(* IEC 61131-3 sources: ironplc-benchmarks/compat_out (part 133) *)

(* revision History
hm	19. jan.2007	rev 1.1
	changed outputs to real to avoid overflow of integer
	added offset for better cascading of scale functions

hm	6. jan. 2008	rev 1.2
	improved performance

hm	26. oct. 2008	rev 1.3
	code optimization

hm	3. nov. 2008	rev 1.4
	used wrong factor in formula

*)
END_FUNCTION

(* @NESTEDCOMMENTS := 'Yes' *)
(* @PATH := '\/Engineering\/signal processing' *)
(* @OBJECTFLAGS := '0, 8' *)
(* @SYMFILEFLAGS := '2048' *)
FUNCTION SCALE_D : REAL
VAR_INPUT
	X : DWORD;
	I_LO : DWORD;
	I_HI : DWORD;
	O_LO : REAL;
	O_HI : REAL;
END_VAR

(*
version 1.2	11. jan. 2011
programmer 	hugo
tested by		oscat

Scale_D is used to translate and scale a DWORD input x to a real output.
the input is limited to I_LO <= X <= I_HI.

*)

(* @END_DECLARATION := '0' *)
IF I_HI = I_LO THEN
	SCALE_D := O_LO;
ELSE
	SCALE_D := (O_HI - O_LO) / DWORD_TO_REAL(I_HI - I_LO) * DWORD_TO_REAL(LIMIT(I_LO, X, I_HI) - I_LO) + O_LO;
END_IF;

(* revision history
hm	18. may. 2008	rev 1.0
	original version

hm	13. nov. 2008	rev 1.1
	corrected formula for negative gradient

hm	11. jan 2011	rev 1.2
	avoid division by 0
*)
END_FUNCTION

(* @NESTEDCOMMENTS := 'Yes' *)
(* @PATH := '\/Engineering\/signal processing' *)
(* @OBJECTFLAGS := '0, 8' *)
(* @SYMFILEFLAGS := '2048' *)
FUNCTION SCALE_R : REAL
VAR_INPUT
	X : REAL;
	I_LO : REAL;
	I_HI : REAL;
	O_LO : REAL;
	O_HI : REAL;
END_VAR

(*
version 1.2	11. jan. 2011
programmer 	hugo
tested by		oscat

Scale_R is used to translate and scale a REAL input x to a real output.
the input is limited to I_LO <= X <= I_HI.

*)

(* @END_DECLARATION := '0' *)
IF I_LO = I_HI THEN
	SCALE_R := O_LO;
ELSE
	SCALE_R := (O_HI - O_LO) / (I_HI - I_LO) * (LIMIT(I_LO, X, I_HI) - I_LO) + O_LO;
END_IF;

(* revision history
hm	18. may. 2008	rev 1.0
	original version

hm	13. nov. 2008	rev 1.1
	corrected formula for negative gradient

hm	11. jan 2011	rev 1.2
	avoid division by 0

*)
END_FUNCTION

(* @NESTEDCOMMENTS := 'Yes' *)
(* @PATH := '\/Engineering\/signal processing' *)
(* @OBJECTFLAGS := '0, 8' *)
(* @SYMFILEFLAGS := '2048' *)
FUNCTION SCALE_X2 : REAL
VAR_INPUT
	IN1: BOOL;
	IN2: BOOL;
	K : REAL;
	O : REAL;
END_VAR
VAR_INPUT (* CONSTANT *)
	IN1_MIN: REAL;
	IN1_MAX: REAL := 1000.0;
	IN2_MIN: REAL;
	IN2_MAX: REAL := 1000.0;
END_VAR

(*
version 1.1	26. oct. 2008
programmer 	hugo
tested by		tobias

	this functiob block can scale up to two inputs.
	the input can select between two values with true or false.
	the summed output is then scaled by an scale input K and a offset O can be added to the output.
	the min and max input configurations can be edited in the cfc editor by double clicking the symbol body.

*)

(* @END_DECLARATION := '0' *)
SCALE_X2 := (SEL(IN1, IN1_MIN, IN1_MAX)+ SEL(IN2, IN2_MIN, IN2_MAX)) * k + o;

(* revision history
hm	19. jan, 2007	rev 1.0
	original version

hm	26. oct. 2008	rev 1.1
	code optimized

*)
END_FUNCTION

(* @NESTEDCOMMENTS := 'Yes' *)
(* @PATH := '\/Engineering\/signal processing' *)
(* @OBJECTFLAGS := '0, 8' *)
(* @SYMFILEFLAGS := '2048' *)
FUNCTION SCALE_X4 : REAL
VAR_INPUT
	IN1: BOOL;
	IN2: BOOL;
	IN3: BOOL;
	IN4: BOOL;
	K : REAL;
	O : REAL;
END_VAR
VAR_INPUT (* CONSTANT *)
	IN1_MIN: REAL;
	IN1_MAX: REAL := 1000.0;
	IN2_MIN: REAL;
	IN2_MAX: REAL := 1000.0;
	IN3_MIN: REAL;
	IN3_MAX: REAL := 1000.0;
	IN4_MIN: REAL;
	IN4_MAX: REAL := 1000.0;
END_VAR

(*
version 1.1	26. oct. 2008
programmer 	hugo
tested by		tobias

	this function can scale up to 4 inputs.
	the input can select between two values with true or false.
	the summed output is then scaled by an scale input K and a offset O can be added to the output.
	the min and max input configurations can be edited in the cfc editor by double clicking the symbol body.

*)

(* @END_DECLARATION := '0' *)
SCALE_X4 := (SEL(IN1,IN1_MIN, IN1_MAX) + SEL(IN2, IN2_MIN, IN2_MAX)+SEL(IN3, IN3_MIN, IN3_MAX)+ SEL(IN4, IN4_MIN, IN4_MAX)) * k + o;

(* revision history
hm	19. jan. 2008	rev 1.0
	original version

hm	26. oct. 2008	rev 1.1
	optimized code
*)
END_FUNCTION

(* @NESTEDCOMMENTS := 'Yes' *)
(* @PATH := '\/Engineering\/signal processing' *)
(* @OBJECTFLAGS := '0, 8' *)
(* @SYMFILEFLAGS := '2048' *)
FUNCTION SCALE_X8 : REAL
VAR_INPUT
	in1: BOOL;
	in2: BOOL;
	in3: BOOL;
	in4: BOOL;
	in5: BOOL;
	in6: BOOL;
	in7: BOOL;
	in8: BOOL;
	K : REAL;
	O : REAL;
END_VAR
VAR_INPUT (* CONSTANT *)
	in1_min: REAL;
	in1_max: REAL := 1000.0;
	in2_min: REAL;
	in2_max: REAL := 1000.0;
	in3_min: REAL;
	in3_max: REAL := 1000.0;
	in4_min: REAL;
	in4_max: REAL := 1000.0;
	in5_min: REAL;
	in5_max: REAL := 1000.0;
	in6_min: REAL;
	in6_max: REAL := 1000.0;
	in7_min: REAL;
	in7_max: REAL := 1000.0;
	in8_min: REAL;
	in8_max: REAL := 1000.0;
END_VAR

(*
version 1.2	24. jan. 2009
programmer 	hugo
tested by	oscat

this function can scale up to 4 inputs.
the input can select between two values with true or false.
the summed output is then scaled by an scale input K and a offset O can be added to the output.
the min and max input configurations can be edited in the cfc editor by double clicking the symbol body.

*)

(* @END_DECLARATION := '0' *)
SCALE_X8 := (SEL(IN1,IN1_MIN, IN1_MAX)+ SEL(IN2,IN2_MIN, IN2_MAX)+SEL(IN3,IN3_MIN, IN3_MAX)+ SEL(IN4,IN4_MIN, IN4_MAX)
				+SEL(IN5,IN5_MIN, IN5_MAX)+ SEL(IN6,IN6_MIN, IN6_MAX)+SEL(IN7,IN7_MIN, IN7_MAX)+ SEL(IN8,IN8_MIN, IN8_MAX)) * k + o;

(* revision history
hm	19. jan. 2008	rev 1.0
	original version

hm	26. oct. 2008	rev 1.1
	optimized code

hm	24. jan. 2008	rev 1.2
	corrected error in formula
*)
END_FUNCTION

(* @NESTEDCOMMENTS := 'Yes' *)
(* @PATH := '\/Engineering\/signal processing' *)
(* @OBJECTFLAGS := '0, 8' *)
(* @SYMFILEFLAGS := '2048' *)
FUNCTION_BLOCK SEL2_OF_3
VAR_INPUT
	IN1 : REAL;
	IN2 : REAL;
	IN3 : REAL;
	D : REAL;
END_VAR
VAR_OUTPUT
	Y : REAL;
	W : INT;
	E : BOOL;
END_VAR
VAR
	D12: BOOL;
	D23: BOOL;
	D31: BOOL;
END_VAR

(*
	version 1.1	10. mar. 2009
	programmer 	oscat
	tested BY		oscat

SEL2_OF_3 checks if 3 input Signals are within a distance D from each other and calculates the average of the 3 inputs do not offset more than D from each other.
If 1 input is more than D greater or smaller than any other input it will be ignored and the average will be calcualted from the remaining 2 Inputs.
In the case the Output is only calculated from 2 Inputs a Warning Output W will display the Number of the discarded Input. if none of the 3 Inputs are within the allowed Delata D from each other,
an Error Output E is set True and the last valid Output will remain active until at least 2 Inputs are within a valid Range from each other.

*)

(* @END_DECLARATION := '0' *)
D12 := ABS(IN1-IN2) <= D;
D23 := ABS(IN2-IN3) <= D;
D31 := ABS(IN3-IN1) <= D;

IF (D12 AND D23) OR (D12 AND D31) OR (D23 AND D31) THEN
	(* all 3 inputs are valid *)
	Y := (IN1 + IN2 + IN3) * 0.333333333333;
	E := FALSE;
	W := 0;
ELSIF D12 THEN
	(* only inut 1 and 2 are valid *)
	Y := (In1 + IN2) * 0.5;
	E := FALSE;
	W := 3;
ELSIF D23 THEN
	(* only inut 2 and 3 are valid *)
	Y := (In2 + IN3) * 0.5;
	E := FALSE;
	W := 1;
ELSIF D31 THEN
	(* only inut 3 and 1 are valid *)
	Y := (In3 + IN1) * 0.5;
	E := FALSE;
	W := 2;
ELSE
	(* no calculation possible *)
	E := TRUE;
	W := 4;
END_IF;

(* revision history
hm	18. may 2008	rev 1.0
	original version

hm	10. mar. 2009	rev 1.1
	improved code
*)
END_FUNCTION_BLOCK

(* @NESTEDCOMMENTS := 'Yes' *)
(* @PATH := '\/Engineering\/signal processing' *)
(* @OBJECTFLAGS := '0, 8' *)
(* @SYMFILEFLAGS := '2048' *)
FUNCTION_BLOCK SEL2_OF_3B
VAR_INPUT
	IN1 : BOOL;
	IN2 : BOOL;
	IN3 : BOOL;
	TD : TIME;
END_VAR
VAR_OUTPUT
	Q : BOOL;
	W : BOOL;
END_VAR
VAR
	TDEL : TON;
END_VAR

(*
	version 1.0	19. may. 2008
	programmer 	oscat
	tested BY		oscat

SEL2_OF_3B is used to connect 3 binary sensors to one signal. the output Q reflects the state of at least two inputs.
if two or more of the 3 inputs ate TRUE then Q will be TRUE and if two or more of the three inputs are FALSE then Q will be false.
the main putrpose is the connection of 3 redundant binary sensors.
The output W will be active when one of the 3 inputs is of different state.
to avoid flickering while the sensors are switching the output W will become active after a programmed delay of TD.

*)

(* @END_DECLARATION := '0' *)
Q := (IN1 AND IN2) OR (IN1 AND IN3) OR (IN2 AND IN3);
TDEL(IN := (in1 XOR in2) OR (in1 XOR in3) OR (in2 XOR in3), PT := TD);
W := TDEL.Q;

(* revision history
hm		19. may 2008	rev 1.0
	original version

*)
END_FUNCTION_BLOCK

(* @NESTEDCOMMENTS := 'Yes' *)
(* @PATH := '\/Engineering\/signal processing' *)
(* @OBJECTFLAGS := '0, 8' *)
(* @SYMFILEFLAGS := '2048' *)
FUNCTION_BLOCK SH
VAR_INPUT
	in : REAL;
	CLK : BOOL;
END_VAR
VAR_OUTPUT
	out : REAL;
	trig : BOOL;
END_VAR
VAR
	edge : BOOL;
END_VAR

(*
version 1.1	16 jan 2007
programmer 	hugo
tested by		tobias

this sample and hold module samples an input at the rising edge of clk an stores it in out.
the out stays stable until the next rising clk edge appears.
a trigger output as active for one cycle when the output was updated.

*)
(* @END_DECLARATION := '0' *)
IF clk AND NOT edge THEN
	out := in;
	trig := TRUE;
ELSE;
	trig := FALSE;
END_IF;
edge := clk;

(* revision history

hm 16.1.2007	rev 1.1
	added trig output

*)
END_FUNCTION_BLOCK

(* @NESTEDCOMMENTS := 'Yes' *)
(* @PATH := '\/Engineering\/signal processing' *)
(* @OBJECTFLAGS := '0, 8' *)
(* @SYMFILEFLAGS := '2048' *)
FUNCTION_BLOCK SH_1
VAR_INPUT
	in : REAL;
	PT : TIME;
END_VAR
VAR_OUTPUT
	out : REAL;
	Trig : BOOL;
END_VAR
VAR
	last : TIME;
	tx: TIME;
END_VAR

(*
version 1.2	17 sep 2007
programmer 	hugo
tested by		tobias

this sample and hold module samples an input every PT seconds.
after a ample is taken the output Trig will be active for one cycle.

*)
(* @END_DECLARATION := '0' *)
(* read system time *)
tx := DWORD_TO_TIME(T_PLC_MS());

IF tx - last >= PT THEN
	last := tx;
	out := in;
	trig := TRUE;
ELSE
	trig := FALSE;
END_IF;

(* revision history

HM	6.1.2007	rev 1.1
	added trig output

HM	17.9.2007	rev 1.2
	replaced time() with T_PLC_MS() for compatibility reasons
*)

END_FUNCTION_BLOCK

(* @NESTEDCOMMENTS := 'Yes' *)
(* @PATH := '\/Engineering\/signal processing' *)
(* @OBJECTFLAGS := '0, 8' *)
(* @SYMFILEFLAGS := '2048' *)
FUNCTION_BLOCK SH_2
VAR_INPUT
	in : REAL;
	PT : TIME;
	N : INT := 16;
	disc : INT;
END_VAR
VAR_OUTPUT
	out : REAL;
	trig : BOOL;
	avg : REAL;
	high: REAL;
	low: REAL;
END_VAR
VAR
	M : INT;
	buf : ARRAY[0..15] OF REAL;
	buf2 : ARRAY[0..15] OF REAL;
	last : TIME;
	i : INT;
	start: INT;
	temp: REAL;
	stop: INT;
	tx: TIME;
	d2: INT;
END_VAR

(*
version 1.6	10. mar. 2009
programmer 	hugo
tested by		tobias

this sample and hold module samples an input every PT seconds.
this sample and hold also does avg and other calculations with the input data.
an average is calculated over N samples while for this calculation disc samples are discarded,
disc = 0 all samples are averaged,
if disc = 1 the lowest value is ignored,
if disc = 2 the lowest and highest values are ignored,
and so on.....

*)
(* @END_DECLARATION := '0' *)
(* read system time *)
tx := DWORD_TO_TIME(T_PLC_MS());
d2 := SHR(disc,1);

IF tx - last >= PT THEN
	last := tx;
	trig := TRUE;

	(* limit M to 0..16 *)
	M := LIMIT(1,N,16);

	(* edge detected lets take the sample *)
	FOR i := M - 1 TO 1 BY -1 DO buf2[i] := buf2[i-1]; END_FOR;
	buf2[0] := in;
	out := in;
	buf := buf2;

	(* sort the ARRAY lowest value AT 0 *)
	FOR start := 0 TO M - 2 DO
		FOR i := start+1 TO M - 1 DO
			IF buf[start] > buf[i] THEN
				temp := buf[start];
				buf[start] := buf[i];
				buf[i] := temp;
			END_IF;
		END_FOR;
	END_FOR;

	(* any calculation with the samples is here *)
	stop := M - 1 - d2;
	start := d2;
	IF NOT even(disc) THEN start := start + 1; END_IF;
	avg := 0;
	FOR i := start TO stop DO avg := avg + buf[i]; END_FOR;
	avg := avg / INT_TO_REAL(stop - start +1);
	low := buf[start];
	high := buf[stop];
ELSE
	Trig := FALSE;
END_IF;

(* revision history
hm 20. jan. 2007	rev 1.1
	added input N to specify the amout of samples for average and high low calculations
	added trig output

hm 10. sep. 2007 	rev 1.2
	an error would be generated if N was set to 0, now n is forced to1 if set to 0.
	index was out of array.

hm	17. sep. 2007	rev 1.3
	replaced time() with t_plc_ms() for compatibility reasons

hm	6. jan. 2008	rev 1.4
	improved performance

hm	14. jun. 2008	rev 1.5
	set default for input N = 16

hm	10. mar. 2009	rev 1.6
	added type conversion for compatibility reasons

*)
END_FUNCTION_BLOCK

(* @NESTEDCOMMENTS := 'Yes' *)
(* @PATH := '\/Engineering\/signal processing' *)
(* @OBJECTFLAGS := '0, 8' *)
(* @SYMFILEFLAGS := '2048' *)
FUNCTION_BLOCK SH_T
VAR_INPUT
	IN : REAL;
	E : BOOL;
END_VAR
VAR_OUTPUT
	OUT : REAL;
END_VAR

(*
version 1.1	18. oct. 2008
programmer 	hugo
tested by	oscat

this sample and hold module samples an input while en is high.
during the high time of en the output follows in.
the out stays stable until the en goes high again.
*)
(* @END_DECLARATION := '0' *)
IF E THEN out := in; END_IF;

(* revision history
hm	1. sep. 2006	rev 1.0
	original version

hm	18. oct. 2008	rev 1.1
	changed input en to e for compatibility reasons

*)
END_FUNCTION_BLOCK

(* @NESTEDCOMMENTS := 'Yes' *)
(* @PATH := '\/Engineering\/signal processing' *)
(* @OBJECTFLAGS := '0, 8' *)
(* @SYMFILEFLAGS := '2048' *)
FUNCTION STAIR : REAL
VAR_INPUT
	X : REAL;
	D : REAL;
END_VAR

(*
version 1.4	10. mar. 2009
programmer 	oscat
tested by		tobias

the function stair converts an anlog input signal to a staircase like output.
D is the step width for the output signal.
if D = 0 then the output follows the input without a chage.
*)
(* @END_DECLARATION := '0' *)
IF D > 0.0 THEN
	STAIR := DINT_TO_REAL(REAL_TO_DINT(X / D)) * D;
ELSE
	STAIR := X;
END_IF;

(* revision history
hm	28 jan 2007		rev 1.0
	original version

hm	27 dec 2007		rev 1.1
	changed code for better performance

hm	6. jan 2008		rev 1.2
	further performance improvement

hm	26. oct. 2008		rev 1.3
	optimized code

hm	10. mar. 2009	rev 1.4
	real constants updated to new systax using dot

*)
END_FUNCTION

(* @NESTEDCOMMENTS := 'Yes' *)
(* @PATH := '\/Engineering\/signal processing' *)
(* @OBJECTFLAGS := '0, 8' *)
(* @SYMFILEFLAGS := '2048' *)
FUNCTION_BLOCK STAIR2
VAR_INPUT
	X : REAL;
	D : REAL;
END_VAR
VAR_OUTPUT
	Y: REAL;
END_VAR

(*
version 1.4	10. mar. 2009
programmer 	hugo
tested by		oscat

the function stair2 converts an anlog input signal to a staircase like output.
D is the step width for the output signal. the output will use D as a hysteresis for a stairchange.
if D = 0 then the output follows the input without a chage.
*)
(* @END_DECLARATION := '0' *)
IF D > 0.0 THEN
	IF X >= Y + D OR X <= Y - D THEN Y := FLOOR(X/D) * D; END_IF;
ELSE
	Y := X;
END_IF;

(* revision history
hm	28 jan 2007		rev 1.0
	original version

hm	27. dec 2007	rev 1.1
	changed code for better performance

hm	30. jun. 2008	rev 1.2
	added type conversions to avoid warnings under codesys 3.0

ks	26. oct. 2008	rev 1.3
	improved code

hm	10. mar. 2009	rev 1.4
	real constants updated to new systax using dot

*)
END_FUNCTION_BLOCK

(* @NESTEDCOMMENTS := 'Yes' *)
(* @PATH := '\/Engineering\/signal processing' *)
(* @OBJECTFLAGS := '0, 8' *)
(* @SYMFILEFLAGS := '2048' *)
FUNCTION_BLOCK TREND
VAR_INPUT
	X : REAL;
END_VAR
VAR_OUTPUT
	Q : BOOL;
	TU : BOOL;
	TD : BOOL;
	D : REAL;
END_VAR
VAR
	last_X: REAL;
END_VAR

(*
version 1.0	21. aug. 2009
programmer 	hugo
tested by		oscat

trend analyses the trend of a input signal.
The Output Q is True if the input X is >= last_X and is false if the input X is <= last_X
in addition to the trend the output TU will be high for one cycle to signal a rising of the input value X
and  TD will signal a decreasing value on the input X.
in case of a change the output D will show the delta of the input to the last input value.

*)
(* @END_DECLARATION := '0' *)
TU := X > last_X;
TD := X < last_X;
Q := TU OR TD;
D := X - LAST_X;

last_X := X;

(* revision history
hm	21. aug. 2009	rev 1.0
	original version

*)

END_FUNCTION_BLOCK

(* @NESTEDCOMMENTS := 'Yes' *)
(* @PATH := '\/Engineering\/signal processing' *)
(* @OBJECTFLAGS := '0, 8' *)
(* @SYMFILEFLAGS := '2048' *)
FUNCTION_BLOCK TREND_DW
VAR_INPUT
	X : DWORD;
END_VAR
VAR_OUTPUT
	Q : BOOL;
	TU : BOOL;
	TD : BOOL;
	D : DWORD;
END_VAR
VAR
	last_X: DWORD;
END_VAR

(*
version 1.2	14. mar. 2009
programmer 	hugo
tested by		oscat

trend_DW analyses the trend of a input signal.
The Output Q is True if the input X is >= last_X and is false if the input X is <= last_X
in addition to the trend the output TU will be high for one cycle to signal a rising of the input value X
and  TD will signal a decreasing value on the input X.
in case of a change the output D will show the delta of the input to the last input value.

*)
(* @END_DECLARATION := '0' *)
IF X > last_X THEN
	TU := TRUE;
	TD := FALSE;
	D := X - last_X;
	Q := TRUE;
ELSIF X < last_X THEN
	TD := TRUE;
	TU := FALSE;
	D := last_X - X;
	Q := FALSE;
ELSE
	TU := FALSE;
	TD := FALSE;
	D := 0;
END_IF;
last_X := X;

(* revision history
hm	21. nov. 2008	rev 1.0
	original version

hm	20. feb. 2009	rev 1.1
	added outputs TU, TD and D

hm	14. mar. 2009	rev 1.2
	removed double assignments

*)

END_FUNCTION_BLOCK

(* @NESTEDCOMMENTS := 'Yes' *)
(* @PATH := '\/Engineering\/signal processing' *)
(* @OBJECTFLAGS := '0, 8' *)
(* @SYMFILEFLAGS := '2048' *)
FUNCTION WORD_TO_RANGE : REAL
VAR_INPUT
	X : WORD;
	low : REAL;
	high : REAL;
END_VAR

(*
version 1.1	10. mar. 2009
programmer 	hugo
tested by		tobias

Word_to_Range converts a Byte into a real between low and high.

*)
(* @END_DECLARATION := '0' *)
WORD_TO_RANGE := (high - low) * WORD_TO_REAL(X) * 0.00001525902189669640 + low;

(* revision history
hm	9. jan 2008	rev 1.0
	original version

hm	10. mar. 2009	rev 1.1
	improved code
*)

END_FUNCTION

(* @NESTEDCOMMENTS := 'Yes' *)
(* @PATH := '\/List Processing' *)
(* @OBJECTFLAGS := '0, 8' *)
(* @SYMFILEFLAGS := '2048' *)
FUNCTION LIST_ADD : BOOL
VAR_INPUT
	SEP : BYTE;
	INS : STRING[LIST_LENGTH];
END_VAR
VAR_IN_OUT
	LIST : STRING[LIST_LENGTH];
END_VAR
VAR
	sx : STRING[1];
END_VAR

(*
version 2.0		21. mar. 2011
programmer 	hugo
tested by		kurt

LIST_ADD h�ngt ein weiteres element ans ende einer liste.
die liste liegt als string von elementen vor die mit den zeichen SEP am anfang makiert sind.

*)
(* @END_DECLARATION := '0' *)
sx := CHR_TO_STRING(SEP);			(* convert separation character to string *)
INS := CONCAT(sx, INS);					(* start element with separation character *)

IF LEN(LIST) + LEN(INS) > LIST_LENGTH THEN
	LIST_ADD := FALSE;					(* return false if element does not fit *)
ELSE
	LIST := CONCAT(LIST, INS);
	LIST_ADD := TRUE;
END_IF;

(* revision histroy

hm	21. mar. 2011	rev 2.0
	original release
*)

END_FUNCTION

(* @NESTEDCOMMENTS := 'Yes' *)
(* @PATH := '\/List Processing' *)
(* @OBJECTFLAGS := '0, 8' *)
(* @SYMFILEFLAGS := '2048' *)
FUNCTION LIST_CLEAN : BOOL
VAR_INPUT
	SEP : BYTE;
END_VAR
VAR_IN_OUT
	LIST : STRING[LIST_LENGTH];
END_VAR
VAR
	pt : REF_TO ARRAY[1..LIST_LENGTH] OF BYTE;
	read : INT := 1;
	write : INT := 1;
	last: BYTE;
	c: BYTE;
END_VAR

(*
version 2.0	21. mar. 2011
programmer 	hugo
tested by		oscat

LIST_CLEAN bereinigt eine liste von leeren Elementen.
die liste liegt als string von elementen vor die mit den zeichen SEP am anfang markiert sind.

*)
(* @END_DECLARATION := '0' *)
pt := REF(LIST);

FOR read := 1 TO LIST_LENGTH DO
	c := pt^[read];								(* read character from list *)
	IF c = 0 THEN EXIT;						(* exit the loop if character definbes end of string *)
	ELSIF c <> SEP OR sep <> last THEN	(* copy element from read to write position unless a double sep character is present *)
		pt^[write] := c;
		write := write + 1;
	END_IF;
	last := c;									(* remember last character *)
END_FOR;

IF last = SEP THEN write := write - 1; END_IF;		(* if last character is sep then delete empty element at end *)
IF write <= STRING_LENGTH THEN pt^[write] := 0;	 END_IF;		(* terminate string with 0 *)

LIST_CLEAN := TRUE;						(* retrun TRUE *)

(* revision histroy
hm	28. jun. 2008	rev 1.0
	original release

hm	19. jan. 2011	rev 1.1
	changed STRING[255] to STRING[LIST_LENGTH]

hm	21. mar. 2011	rev 2.0
	all elements start with SEP

*)

END_FUNCTION

(* @NESTEDCOMMENTS := 'Yes' *)
(* @PATH := '\/List Processing' *)
(* @OBJECTFLAGS := '0, 8' *)
(* @SYMFILEFLAGS := '2048' *)
FUNCTION LIST_GET : STRING[LIST_LENGTH]
VAR_INPUT
	SEP : BYTE;
	POS : INT;
END_VAR
VAR_IN_OUT
	LIST : STRING[LIST_LENGTH];
END_VAR
VAR
	i : INT := 1;
	o : INT := 1;
	pt : REF_TO ARRAY[1..LIST_LENGTH] OF BYTE;
	po : REF_TO ARRAY[1..LIST_LENGTH] OF BYTE;
	cnt: INT := 0;
	c: BYTE;
END_VAR

(*
version 2.0	21. mar. 2011
programmer 	hugo
tested by		oscat

LIST_GET liefert das element an der stelle pos einer liste.
die liste liegt als string von elementen vor die mit den zeichen SEP am anfang makiert sind.

*)
(* @END_DECLARATION := '0' *)
pt := REF(LIST);							(* load pointers *)
po := REF(LIST_GET);

REPEAT
	c := pt^[i];
	IF cnt = pos THEN						(* copy element to output string *)
		IF c = SEP  THEN EXIT; END_IF;		(* next element stop copy and finish *)
		po^[o] := c;
		o := o + 1;
	ELSIF c = SEP THEN
		cnt := cnt + 1;
	END_IF;
	i := i + 1;
UNTIL
	(i = LIST_LENGTH) OR (c = 0)
END_REPEAT;
po^[o] := 0;						(* close the output string *)

(* revision histroy
hm	20. jun. 2008	rev 1.0
	original release

hm	19. jan. 2011	rev 1.1
	changed STRING[255] to strring(LIST_LENGTH)

hm	21. mar. 2011	rev 2.0
	all list elements start with SEP
*)

END_FUNCTION

(* @NESTEDCOMMENTS := 'Yes' *)
(* @PATH := '\/List Processing' *)
(* @OBJECTFLAGS := '0, 8' *)
(* @SYMFILEFLAGS := '2048' *)
FUNCTION LIST_INSERT : BOOL
VAR_INPUT
	SEP : BYTE;
	POS : INT;
	INS : STRING[LIST_LENGTH];
END_VAR
VAR_IN_OUT
	LIST : STRING[LIST_LENGTH];
END_VAR
VAR
	pt : REF_TO ARRAY[1..LIST_LENGTH] OF BYTE;
	read : INT := 1;
	cnt : INT := 1;
	sx : STRING[1];
END_VAR

(*
version 2.0	21. mar. 2011
programmer 	hugo
tested by		oscat

LIST_INSERT setzt ein element an der stelle pos in eine liste ein.
die liste liegt als string von elementen vor die mit den zeichen SEP am anfang markiert sind.

*)
(* @END_DECLARATION := '0' *)
(* load pointers *)
pt := REF(LIST);

IF LEN(ins) + 1 + LEN(LIST) > LIST_LENGTH THEN
	LIST_INSERT := FALSE;
ELSE
	LIST_INSERT := TRUE;
	(* search for position *)
	WHILE read < LIST_LENGTH DO
		IF cnt >= POS THEN
			sx := CHR_TO_STRING(SEP);
			INS := CONCAT(sx, INS);
			LIST := INSERT(LIST, INS, read - 1);
			LIST_INSERT := TRUE;
			RETURN;
		END_IF;
		IF pt^[read]  = 0 THEN				(* list is too short add empty element *)
			pt^[read] := SEP;
			pt^[read + 1] := 0;
		END_IF;
		read := read + 1;
		IF pt^[read] = SEP OR pt^[read] = 0 THEN cnt := cnt + 1; END_IF;
	END_WHILE;
END_IF;

(* revision histroy
hm	28. jun. 2008	rev 1.0
	original release

hm	17. dec. 2008	rev 1.1
	changes name of function chr to chr_to_string

hm	19. jan. 2011	rev 1.2
	changed STRING[255] to STRING[LIST_LENGTH]

hm	21. mar. 2011	rev 2.0
	all list elements start with SEP

*)

END_FUNCTION

(* @NESTEDCOMMENTS := 'Yes' *)
(* @PATH := '\/List Processing' *)
(* @OBJECTFLAGS := '0, 8' *)
(* @SYMFILEFLAGS := '2048' *)
FUNCTION LIST_LEN : INT
VAR_INPUT
	SEP : BYTE;
END_VAR
VAR_IN_OUT
	LIST : STRING[LIST_LENGTH];
END_VAR
VAR
	pt : REF_TO ARRAY[1..LIST_LENGTH] OF BYTE;
	pos: INT := 1;
	c: BYTE;
END_VAR

(*
version 2.0	21. mar. 2011
programmer 	hugo
tested by		oscat

LIST_LEN liefert die anzahl der elemente einer liste.
die liste liegt als string von elementen vor die mit den zeichen SEP am anfang markiert sind.

*)
(* @END_DECLARATION := '0' *)
pt := REF(LIST);
LIST_LEN := 0;
REPEAT
	c := pt^[pos];
	IF c = SEP THEN LIST_LEN := LIST_LEN + 1; END_IF;
	pos := pos + 1;
UNTIL
	c = 0 OR pos > LIST_LENGTH
END_REPEAT;

(* revision histroy
hm	25. jun. 2008	rev 1.0
	original release

hm	16. oct. 2008	rev 1.1
	fixed a problem where list_len would only work up to LIST_LENGTH

hm	19. jan. 2001	rev 1.2
	changed STRING[255] to STRING[LIST_LENGTH]

hm	21. mar. 2011	rev 2.0
	all list elements start with SEP

*)

END_FUNCTION

(* @NESTEDCOMMENTS := 'Yes' *)
(* @PATH := '\/List Processing' *)
(* @OBJECTFLAGS := '0, 8' *)
(* @SYMFILEFLAGS := '2048' *)
FUNCTION_BLOCK LIST_NEXT
VAR_INPUT
	SEP : BYTE;
	RST : BOOL;
END_VAR
VAR_IN_OUT
	LIST : STRING[LIST_LENGTH];
END_VAR
VAR_OUTPUT
	LEL : STRING[LIST_LENGTH];
	NUL : BOOL;
END_VAR
VAR
	pos : INT := 1;
	pt : REF_TO ARRAY[1..LIST_LENGTH] OF BYTE;
	po : REF_TO ARRAY[1..LIST_LENGTH] OF BYTE;
	c: BYTE;
	write: INT;
END_VAR

(*
version 2.0	21. mar. 2011
programmer 	hugo
tested by		oscat

LIST_NEXT retrieves the next element of a list, starting from element 1 after reset or first init.
when the end of the lisat is reached a '' empty string is returned and NUL is set to true.
die liste liegt als string von elementen vor die mit den zeichen SEP am anfang markiert sind.

*)
(* @END_DECLARATION := '0' *)
pt := REF(LIST);
po := REF(LEL);

IF rst THEN
	pos := 1;
END_IF;

IF pt^[pos] = 0 OR pos = LIST_LENGTH THEN
	LEL := '';
	NUL := TRUE;
ELSE
	NUL := FALSE;
	write := 1;
	FOR pos := pos + 1 TO LIST_LENGTH DO
		c := pt^[pos];
		IF c = 0 OR c = SEP THEN
			po^[write] := 0;
			RETURN;
		ELSE
			po^[write] := pt^[pos];
			write := write + 1;
		END_IF;
	END_FOR;
END_IF;

(* revision histroy
hm	25. jun. 2008	rev 1.0
	original release

hm	19. jan. 2011	rev 1.1
	changed STRING[255] to STRING[LIST_LENGTH]

hm	21. mar. 2011	rev 2.0
	all elements start with SEP

*)

END_FUNCTION_BLOCK

(* @NESTEDCOMMENTS := 'Yes' *)
(* @PATH := '\/List Processing' *)
(* @OBJECTFLAGS := '0, 8' *)
(* @SYMFILEFLAGS := '2048' *)
FUNCTION LIST_RETRIEVE : STRING[LIST_LENGTH]
VAR_INPUT
	SEP : BYTE;
	POS : INT;
END_VAR
VAR_IN_OUT
	LIST : STRING[LIST_LENGTH];
END_VAR
VAR
	i :	INT;
	o : INT := 1;
	w : INT := 1;
	pt : REF_TO ARRAY[1..LIST_LENGTH] OF BYTE;
	po : REF_TO ARRAY[1..LIST_LENGTH] OF BYTE;
	cnt: INT := 0;
	c: BYTE;
END_VAR

(*
version 2.0		21. mar. 2011
programmer 	hugo
tested by		oscat

LIST_RETRIEVE liefert das element an der stelle pos einer liste und l�scht das element aus der liste.
die liste liegt als string von elementen vor die mit den zeichen SEP separiert sind.

*)
(* @END_DECLARATION := '0' *)
(* load pointers *)
pt := REF(LIST);
po := REF(LIST_RETRIEVE);

IF pos > 0 THEN
	FOR i := 1 TO LIST_LENGTH DO
		c := pt^[i];
		IF c = 0 THEN
			po^[o] := 0;
			IF cnt < pos THEN pt^[w + 1] := 0; ELSE pt^[w] := 0; END_IF;
			RETURN;
		ELSIF cnt = pos AND c <> SEP THEN				(* we have found the element *)
			po^[o] := pt^[i];
			o := o + 1;
		ELSIF cnt >= pos THEN
			pt^[w] := c;
			w := w + 1;
		ELSE
			w := i;
		END_IF;
		IF c = sep THEN cnt := cnt + 1; END_IF;
	END_FOR;
ELSE
	LIST_RETRIEVE := '';
END_IF;

(* revision histroy
hm	28. jun. 2008	rev 1.0
	original release

hm	19. jan. 2011	rev 1.1
	changed STRING[255] to STRING[LIST_LENGTH]

hm	21. mar. 2011	rev 2.0
	all elements start with SEP
*)

END_FUNCTION

(* @NESTEDCOMMENTS := 'Yes' *)
(* @PATH := '\/List Processing' *)
(* @OBJECTFLAGS := '0, 8' *)
(* @SYMFILEFLAGS := '2048' *)
FUNCTION LIST_RETRIEVE_LAST : STRING[LIST_LENGTH]
VAR_INPUT
	SEP : BYTE;
END_VAR
VAR_IN_OUT
	LIST : STRING[LIST_LENGTH];
END_VAR
VAR
	i :	INT;
	last : INT := 1;
	pt : REF_TO ARRAY[1..LIST_LENGTH] OF BYTE;
	c: BYTE;
END_VAR

(*
version 2.0		21. mar. 2011
programmer 	hugo
tested by		oscat

LIST_RETRIEVE_LAST liefert das letzte element einer liste und l�scht das element aus der liste.
die liste liegt als string von elementen vor die mit den zeichen SEP beginnen.

*)
(* @END_DECLARATION := '0' *)
(* load pointers *)
pt := REF(LIST);

(* search position of last element *)
FOR i := 1 TO LIST_LENGTH DO
	c := pt^[i];
	IF c = 0 THEN
		EXIT;
	ELSIF C = SEP THEN
		last := i;
	END_IF;
END_FOR;
(* return last element of list *)
/* LIST_RETRIEVE_LAST := MID(LIST, LIST_LENGTH, last + 1); */
(* terminate list at i *)
pt^[last] := 0;

(* revision histroy
hm	21. mar. 2011	rev 2.0
	new module
*)
END_FUNCTION

(* @NESTEDCOMMENTS := 'Yes' *)
(* @PATH := '\/Logic\/FF edge triggered' *)
(* @OBJECTFLAGS := '0, 8' *)
(* @SYMFILEFLAGS := '2048' *)
FUNCTION_BLOCK COUNT_BR
VAR_INPUT
	SET0 : BOOL;
	IN : BYTE;
	UP : BOOL;
	DN : BOOL;
	STEP : BYTE := 1;
	MX : BYTE := 255;
	RST : BOOL;
END_VAR
VAR_OUTPUT
	CNT : BYTE;
END_VAR
VAR
	last_up: BOOL;
	last_dn: BOOL;
END_VAR

(*
	version 1.0	16 jan 2008
	programmer 	hugo
	tested BY	tobias

Count_BR is a byte counter with independen up and dn inputs. the counter counts from 0 to mx and continues at 0 after is has reached mx
a step input sets the counters stepping width.

*)
(* @END_DECLARATION := '0' *)
IF rst THEN
	cnt := 0;
ELSIF set0 THEN
	cnt := LIMIT(0,in,mx);
ELSIF up AND NOT last_up THEN
	cnt := INT_TO_BYTE(INC(cnt,step,mx));
ELSIF dn AND NOT last_dn THEN
	cnt := INT_TO_BYTE(inc(cnt,-step,mx));
END_IF;
last_up := up;
last_dn := dn;

(* revision history
hm	16. jan 2008	rev 1.0
	original version

*)
END_FUNCTION_BLOCK

(* @NESTEDCOMMENTS := 'Yes' *)
(* @PATH := '\/Logic\/FF edge triggered' *)
(* @OBJECTFLAGS := '0, 8' *)
(* @SYMFILEFLAGS := '2048' *)
FUNCTION_BLOCK COUNT_DR
VAR_INPUT
	SET0 : BOOL;
	IN : DWORD;
	UP : BOOL;
	DN : BOOL;
	STEP : DWORD := 1;
	MX : DWORD := 16#FFFFFFFF;
	RST : BOOL;
END_VAR
VAR_OUTPUT
	CNT : DWORD;
END_VAR
VAR
	last_up: BOOL;
	last_dn: BOOL;
END_VAR

(*
	version 1.1	20. jan. 2011
	programmer 	hugo
	tested BY		tobias

Count_DR is a DWORD counter with independen up and dn inputs. the counter counts from 0 to mx and continues at 0 after is has reached mx
a step input sets the counters stepping width.

*)
(* @END_DECLARATION := '0' *)
IF rst THEN
	cnt := 0;
ELSIF set0 THEN
	cnt := LIMIT(0,in,mx);
ELSIF up AND NOT last_up THEN
	IF STEP > MX - CNT THEN
		CNT := CNT - MX + STEP - 1;
	ELSE
		CNT := CNT + STEP;
	END_IF;
ELSIF dn AND NOT last_dn THEN
	IF STEP > CNT THEN
		CNT := CNT - STEP + MX + 1;
	ELSE
		CNT := CNT - STEP;
	END_IF;
END_IF;
last_up := up;
last_dn := dn;

(* revision history
hm	12. jun 2008	rev 1.0
	original version

hm	20. jan. 2011	rev 1.1
	corrected init value of MX to 16#FFFFFFFF

*)
END_FUNCTION_BLOCK

(* @NESTEDCOMMENTS := 'Yes' *)
(* @PATH := '\/Logic\/FF edge triggered' *)
(* @OBJECTFLAGS := '0, 8' *)
(* @SYMFILEFLAGS := '2048' *)
FUNCTION_BLOCK FF_D2E
VAR_INPUT
	D0 : BOOL;
	D1 : BOOL;
	CLK : BOOL;
	RST : BOOL;
END_VAR
VAR_OUTPUT
	Q0 : BOOL;
	Q1 : BOOL;
END_VAR
VAR
	edge : BOOL;
END_VAR

(*
version 1.3	14. mar. 2009
programmer 	hugo
tested by		oscat

dual D-type flip flop with reset and rising clock trigger

*)

(* @END_DECLARATION := '0' *)
IF rst THEN
	Q0 := FALSE;
	Q1 := FALSE;
ELSIF clk AND NOT edge THEN
	Q0 := D0;
	Q1 := D1;
END_IF;
edge := CLK;

(* revision history
hm	25. dec 2007	rev 1.0
	original version

hm	27. dec 2007	rev 1.1
	changed code for better performance

hm	30. oct. 200	rev 1.2
	deleted unnecessary init with 0

hm	14. mar. 2009	rev 1.3
	removed double assignments

*)

END_FUNCTION_BLOCK

(* @NESTEDCOMMENTS := 'Yes' *)
(* @PATH := '\/Logic\/FF edge triggered' *)
(* @OBJECTFLAGS := '0, 8' *)
(* @SYMFILEFLAGS := '2048' *)
FUNCTION_BLOCK FF_D4E
VAR_INPUT
	D0 : BOOL;
	D1 : BOOL;
	D2 : BOOL;
	D3 : BOOL;
	CLK : BOOL;
	RST : BOOL;
END_VAR
VAR_OUTPUT
	Q0 : BOOL;
	Q1 : BOOL;
	Q2 : BOOL;
	Q3 : BOOL;
END_VAR
VAR
	edge : BOOL;
END_VAR

(*
version 1.3	14. mar. 2009
programmer 	hugo
tested by		oscat

quad D-type flip flop with reset and rising clock trigger

*)

(* @END_DECLARATION := '0' *)
IF rst THEN
	Q0 := FALSE;
	Q1 := FALSE;
	Q2 := FALSE;
	Q3 := FALSE;
ELSIF clk AND NOT edge THEN
	Q0 := D0;
	Q1 := D1;
	Q2 := D2;
	Q3 := D3;
END_IF;
edge := CLK;

(* revision history
hm	4. aug 2006	rev 1.0
	original version

hm	27. dec 2007	rev 1.1
	changed code for better performance

hm	30. oct. 200	rev 1.2
	deleted unnecessary init with 0

hm	14. mar. 2009	rev 1.3
	removed double assignments

*)

END_FUNCTION_BLOCK

(* @NESTEDCOMMENTS := 'Yes' *)
(* @PATH := '\/Logic\/FF edge triggered' *)
(* @OBJECTFLAGS := '0, 8' *)
(* @SYMFILEFLAGS := '2048' *)
FUNCTION_BLOCK FF_DRE
VAR_INPUT
	SET0 : BOOL;
	D : BOOL;
	CLK : BOOL;
	RST : BOOL;
END_VAR
VAR_OUTPUT
	Q : BOOL;
END_VAR
VAR
	edge : BOOL;
END_VAR

(*
version 1.2	30. oct. 2008
programmer 	hugo
tested by	oscat

D-type flip flop with set, reset and rising clock trigger

*)

(* @END_DECLARATION := '0' *)
IF rst OR set0 THEN
	Q := NOT rst;
ELSIF clk AND NOT edge THEN
	Q := D;
END_IF;
edge := CLK;

(* revision history
hm	4. aug 2006		rev 1.0
	original version

hm	27. dec 2007	rev 1.1
	changed code for better performance

hm	30. oct. 2008	rev 1.2
	optimized performance
*)
END_FUNCTION_BLOCK

(* @NESTEDCOMMENTS := 'Yes' *)
(* @PATH := '\/Logic\/FF edge triggered' *)
(* @OBJECTFLAGS := '0, 8' *)
(* @SYMFILEFLAGS := '2048' *)
FUNCTION_BLOCK FF_JKE
VAR_INPUT
	SET0 : BOOL;
	J : BOOL;
	CLK : BOOL;
	K : BOOL;
	RST : BOOL;
END_VAR
VAR_OUTPUT
	Q : BOOL;
END_VAR
VAR
	edge : BOOL;
END_VAR

(*
version 1.2	30. oct. 2008
programmer 	hugo
tested by	oscat

JK-type flip flop with set, reset and rising clock trigger
set and reset are asynchron while the FF is rising edge triggered
J=0 and K=0 and CLK >>> no action
J=1 and K=0 and CLK >>> output = 1
J=0 and K=1 and CLK >>> output = 0
J=1 and K=1 and CLK >>> toggle output

*)

(* @END_DECLARATION := '0' *)
IF rst OR set0 THEN
	Q := NOT rst;
ELSIF clk AND NOT edge THEN
	IF J XOR K THEN Q := J;
	ELSE Q := K XOR Q;
	END_IF;
END_IF;
edge := CLK;

(* revision history
hm	4. aug 2006		rev 1.0
	original version

hm	27. dec 2007	rev 1.1
	changed code for better performance

hm	30. oct. 2008	rev 1.2
	optimized performance
*)
END_FUNCTION_BLOCK

(* @NESTEDCOMMENTS := 'Yes' *)
(* @PATH := '\/Logic\/FF edge triggered' *)
(* @OBJECTFLAGS := '0, 8' *)
(* @SYMFILEFLAGS := '2048' *)
FUNCTION_BLOCK FF_RSE
VAR_INPUT
	CS : BOOL;
	CR : BOOL;
	RST : BOOL;
END_VAR
VAR_OUTPUT
	Q : BOOL;
END_VAR
VAR
	es, er : BOOL;
END_VAR

(*
version 1.0	16. jul. 2008
programmer 	hugo
tested by	oscat

this is a rising edge triggered rs flip flop
a rising edge on CS sets Q = TRUE and a rising edge on CR sets Q = FALSE.
CR has priority over CS.

*)

(* @END_DECLARATION := '0' *)
IF rst THEN
	(* asynchronous reset *)
	Q := FALSE;
ELSIF CR AND NOT er THEN
	(* rising edge on CR *)
	Q := FALSE;
ELSIF CS AND NOT es THEN
	(* rising edge on CS *)
	Q := TRUE;
END_IF;

es := CS;
er := CR;

(* revision history

hm	16. jul. 2008	rev 1.0
	original version

*)

END_FUNCTION_BLOCK

(* @NESTEDCOMMENTS := 'Yes' *)
(* @PATH := '\/Logic\/FF edge triggered' *)
(* @OBJECTFLAGS := '0, 8' *)
(* @SYMFILEFLAGS := '2048' *)
FUNCTION_BLOCK SELECT_8
VAR_INPUT
	E : BOOL;
	SET0 : BOOL;
	IN : BYTE;
	UP : BOOL;
	DN : BOOL;
	RST : BOOL;
END_VAR
VAR_OUTPUT
	Q0, Q1, Q2, Q3, Q4, Q5, Q6, Q7 : BOOL;
	STATE : INT;
END_VAR
VAR
	last_up: BOOL;
	last_dn : BOOL;
END_VAR

(*
	version 1.1	27. feb. 2009
	programmer 	hugo
	tested BY		oscat

select_8 selects one of 8 outputs at any time. the outputscan be selected by up or down keys and an independent anable switches all outouts off if set false

*)
(* @END_DECLARATION := '0' *)
IF rst THEN
	state := 0;
ELSIF set0 THEN
	state := IN;
ELSIF up AND NOT last_up THEN
	state := inc(state,1,7);
ELSIF dn AND NOT last_dn THEN
	state := inc(state,-1,7);
END_IF;
last_UP := UP;
last_DN := DN;

Q0 := FALSE;
Q1 := FALSE;
Q2 := FALSE;
Q3 := FALSE;
Q4 := FALSE;
Q5 := FALSE;
Q6 := FALSE;
Q7 := FALSE;

IF E THEN
	CASE state OF
		0: Q0 := TRUE;
		1: Q1 := TRUE;
		2: Q2 := TRUE;
		3: Q3 := TRUE;
		4: Q4 := TRUE;
		5: Q5 := TRUE;
		6: Q6 := TRUE;
		7: Q7 := TRUE;
	END_CASE;
END_IF;

(* revision history
hm	16. jan 2008	rev 1.0
	original version

hm	27. feb. 2009	rev 1.1
	renamed input en to e
*)
END_FUNCTION_BLOCK

(* @NESTEDCOMMENTS := 'Yes' *)
(* @PATH := '\/Logic\/FF edge triggered' *)
(* @OBJECTFLAGS := '0, 8' *)
(* @SYMFILEFLAGS := '2048' *)
FUNCTION_BLOCK SHR_4E
VAR_INPUT
	SET0 : BOOL;
	D0: BOOL;
	CLK: BOOL;
	RST: BOOL;
END_VAR
VAR_OUTPUT
	Q0: BOOL;
	Q1: BOOL;
	Q2: BOOL;
	Q3: BOOL;
END_VAR
VAR
	trig : R_TRIG;
END_VAR

(*
version 1.1	25. oct. 2008
programmer 	hugo
tested by		tobias

4 bit shift register with reset

*)
(* @END_DECLARATION := '0' *)
(* trig.Q signals a rising edge on clk *)
trig(clk := clk);

IF set0 OR rst THEN
	Q0 := NOT rst;
	Q1 := Q0;
	Q2 := Q0;
	Q3 := Q0;
ELSIF trig.Q THEN
	Q3 := Q2;
	Q2 := Q1;
	Q1 := Q0;
	Q0 := D0;
END_IF;

(* revision history
hm	4. aug. 2006	rev 1.0
	original version

hm	25. oct. 2008	rev 1.1
	optimized code

*)
END_FUNCTION_BLOCK

(* @NESTEDCOMMENTS := 'Yes' *)
(* @PATH := '\/Logic\/FF edge triggered' *)
(* @OBJECTFLAGS := '0, 8' *)
(* @SYMFILEFLAGS := '2048' *)
FUNCTION_BLOCK SHR_4UDE
VAR_INPUT
	SET0 : BOOL;
	D0: BOOL;
	D3: BOOL;
	CLK: BOOL;
	DN : BOOL;
	RST: BOOL;

END_VAR
VAR_OUTPUT
	Q0: BOOL;
	Q1: BOOL;
	Q2: BOOL;
	Q3: BOOL;
END_VAR
VAR
	trig : R_TRIG;
END_VAR

(*
version 1.2	14. mar. 2009
programmer 	hugo
tested by		tobias

4 bit shift register with reset up / down direction input

*)
(* @END_DECLARATION := '0' *)
(* trig.Q signals a rising edge on clk *)
trig(clk := clk);

IF set0 OR rst THEN
	Q0 := NOT RST;
	Q1 := Q0;
	Q2 := Q0;
	Q3 := Q0;
ELSIF trig.Q THEN
	IF dn THEN
		Q0 := Q1;
		Q1 := Q2;
		Q2 := Q3;
		Q3 := D3;
	ELSE
		Q3 := Q2;
		Q2 := Q1;
		Q1 := Q0;
		Q0 := D0;
	END_IF;
END_IF;

(* revision history
hm	4. aug. 2006	rev 1.0
	original version

hm	25. oct. 2008	rev 1.1
	optimized code

hm	14. mar. 2009	rev 1.2
	removed double assignments

*)
END_FUNCTION_BLOCK

(* @NESTEDCOMMENTS := 'Yes' *)
(* @PATH := '\/Logic\/FF edge triggered' *)
(* @OBJECTFLAGS := '0, 8' *)
(* @SYMFILEFLAGS := '2048' *)
FUNCTION_BLOCK SHR_8PLE
VAR_INPUT
	Din : BOOL;
	Dload : BYTE;
	CLK: BOOL;
	UP: BOOL :=1;
	load : BOOL;
	RST: BOOL;
END_VAR
VAR_OUTPUT
	DOut: BOOL;
END_VAR
VAR
	edge : BOOL :=1;
	register : BYTE;
END_VAR

(*
version 1.0	4 aug 2006
programmer 	hugo
tested by	oscat

8 bit shift register with reset and parallel load
the register can shift up or down
it also has a serial input.
the Din input is on Bit0 for up shift and on bit 7 for down shift
the Dout output is on Bit7 for up shift and on bit 0 for down shift
paralle clock is performed clock synchron while a shift is performed first and then the register is reloaded

*)
(* @END_DECLARATION := '0' *)
(* flankenerkennung clk wird high und edge war high reset ist nicht aktiv und set ist nicht aktiv *)
IF CLK AND edge AND NOT rst THEN
	edge := FALSE;	(* flanke wurde erkannt und weitere flankenerkennung wird verhindert bis edge wieder true ist *)
	(* hier ist der code f�r das flankenevent *)
	IF UP THEN						(*shift up *)
		register := SHL(register,1);
		register.0 := Din;
		Dout := register.7;
	ELSE								(* shift down *);
		register := SHR(register,1);
		register.7 := Din;
		Dout := register.0;
	END_IF;
	IF load THEN							(* the byte on Din will be loaded if load = true *)
		register := Dload;
		IF up THEN Dout := register.7; ELSE Dout := register.0; END_IF;
	END_IF;
END_IF;
IF NOT clk THEN edge := TRUE; END_IF;	(* sobald clk wieder low wird warten auf n�chste flanke *)
IF rst THEN									(* wenn reset aktiv dann ausgang r�cksetzen *)
	register := 0;
	Dout := FALSE;
END_IF;

END_FUNCTION_BLOCK

(* @NESTEDCOMMENTS := 'Yes' *)
(* @PATH := '\/Logic\/FF edge triggered' *)
(* @OBJECTFLAGS := '0, 8' *)
(* @SYMFILEFLAGS := '2048' *)
FUNCTION_BLOCK SHR_8UDE
VAR_INPUT
	SET0 : BOOL;
	D0: BOOL;
	D7: BOOL;
	CLK: BOOL;
	DN : BOOL;
	RST: BOOL;
END_VAR
VAR_OUTPUT
	Q0: BOOL;
	Q1: BOOL;
	Q2: BOOL;
	Q3: BOOL;
	Q4: BOOL;
	Q5: BOOL;
	Q6: BOOL;
	Q7: BOOL;
END_VAR
VAR
	trig : R_TRIG;
END_VAR

(*
version 1.2	14. mar. 2009
programmer 	hugo
tested by		tobias

8 bit shift register with reset

*)
(* @END_DECLARATION := '0' *)
(* trig.Q signals a rising edge on clk *)
trig(clk := clk);

IF set0 OR rst THEN
	Q0 := NOT RST;
	Q1 := Q0;
	Q2 := Q0;
	Q3 := Q0;
	Q4 := Q0;
	Q5 := Q0;
	Q6 := Q0;
	Q7 := Q0;
ELSIF trig.Q THEN
	IF dn THEN
		Q0 := Q1;
		Q1 := Q2;
		Q2 := Q3;
		Q3 := Q4;
		Q4 := Q5;
		Q5 := Q6;
		Q6 := Q7;
		Q7 := D7;
	ELSE
		Q7 := Q6;
		Q6 := Q5;
		Q5 := Q4;
		Q4 := Q3;
		Q3 := Q2;
		Q2 := Q1;
		Q1 := Q0;
		Q0 := D0;
	END_IF;
END_IF;

(* revision history
hm	4. aug. 2006	rev 1.0
	original version

hm	25. oct. 2008	rev 1.1
	optimized code

hm	14. mar. 2009	rev 1.2
	removed double assignments

*)
END_FUNCTION_BLOCK

(* @NESTEDCOMMENTS := 'Yes' *)
(* @PATH := '\/Logic\/FF edge triggered' *)
(* @OBJECTFLAGS := '0, 8' *)
(* @SYMFILEFLAGS := '2048' *)
FUNCTION_BLOCK TOGGLE
VAR_INPUT
	CLK : BOOL;
	rst : BOOL;
END_VAR
VAR_OUTPUT
	Q : BOOL;
END_VAR
VAR
	edge : BOOL;
END_VAR

(*
version 1.1	30. oct. 2008
programmer 	hugo
tested by	oscat

toggle flip flop the output changes state with every rising edge of clk.

*)

(* @END_DECLARATION := '0' *)
IF rst THEN
	q := 0;
ELSIF clk AND NOT edge THEN
	Q := NOT Q;
END_IF;
edge := clk;

(* revision history

hm	13.9.2007		rev 1.0
	original version

hm	30. oct. 2008	rev 1.1
	deleted unnecessary init

*)

END_FUNCTION_BLOCK

(* @NESTEDCOMMENTS := 'Yes' *)
(* @PATH := '\/Logic\/FF pulse triggered' *)
(* @OBJECTFLAGS := '0, 8' *)
(* @SYMFILEFLAGS := '2048' *)
FUNCTION_BLOCK LTCH
VAR_INPUT
	D : BOOL;
	L : BOOL;
	RST : BOOL;
END_VAR
VAR_OUTPUT
	Q : BOOL;
END_VAR

(*
version 1.2	30. oct. 2008
programmer 	hugo
tested by	oscat

Transparent Latch with asynchronous reset

*)

(* @END_DECLARATION := '0' *)
(* as long as L is true, the latch is transparent and and change of D is transferred to Q *)
(* of course only when there is no asynchronous reset *)
IF rst THEN				(* if asynchronous reset then Q=0 *)
	Q := FALSE;
ELSIF L THEN			(* latch is transparent *)
	Q := D;
END_IF;

(* revision history
hm	4. aug 2006		rev 1.0
	original version

hm	27. dec 2007	rev 1.1
	changed code for better performance

hm	30. oct. 2008	rev 1.2
	deleted unnecessary init with 0

*)
END_FUNCTION_BLOCK

(* @NESTEDCOMMENTS := 'Yes' *)
(* @PATH := '\/Logic\/FF pulse triggered' *)
(* @OBJECTFLAGS := '0, 8' *)
(* @SYMFILEFLAGS := '2048' *)
FUNCTION_BLOCK LTCH_4
VAR_INPUT
	D0 : BOOL;
	D1 : BOOL;
	D2 : BOOL;
	D3 : BOOL;
	L : BOOL;
	RST : BOOL;
END_VAR
VAR_OUTPUT
	Q0 : BOOL;
	Q1 : BOOL;
	Q2 : BOOL;
	Q3 : BOOL;
END_VAR

(*
version 1.3	14. mar. 2009
programmer 	hugo
tested by		oscat

Quad Transparent Latch with asynchronous reset

*)

(* @END_DECLARATION := '0' *)
(* as long as L is true, the latch is transparent and and change of D is transferred to Q *)
(* of course only when there is no asynchronous reset *)
IF rst THEN			(* if asynchronous reset then Q=0 *)
	Q0 := FALSE;
	Q1 := FALSE;
	Q2 := FALSE;
	Q3 := FALSE;
ELSIF L THEN			(* latch is transparent *)
	Q0 := D0;
	Q1 := D1;
	Q2 := D2;
	Q3 := D3;
END_IF;

(* revision history
hm	4. aug 2006	rev 1.0
	original version

hm	27. dec 2007	rev 1.1
	changed code for better performance

hm	30. oct. 2008	rev 1.2
	deleted unnecessary init with 0

hm	14. mar. 2009	rev 1.3
	removed double assignments

*)
END_FUNCTION_BLOCK

(* @NESTEDCOMMENTS := 'Yes' *)
(* @PATH := '\/Logic\/FF pulse triggered' *)
(* @OBJECTFLAGS := '0, 8' *)
(* @SYMFILEFLAGS := '2048' *)
FUNCTION_BLOCK STORE_8
VAR_INPUT
	Set0 : BOOL;
	D0,D1, D2, D3, D4, D5, D6, D7 : BOOL;
	Clr : BOOL;
	Rst : BOOL;
END_VAR
VAR_OUTPUT
	Q0, Q1, Q2, Q3, Q4, Q5, Q6, Q7 : BOOL;
END_VAR
VAR
	edge: BOOL;
END_VAR

(*
version 1.2	14. mar. 2009
programmer 	hugo
tested by		oscat

Store_4 stores up to 4 boolean inputs until a reset is clearing the outputs.
the respective output is set with a true at the respective input and stays true until a reset is generated.
a set input is used to set all outputs true at the same time, independent of their inputs.
a clear input is used to reset only the lowest priority of the outputs one at a time.
the lowest priority is q3.

*)
(* @END_DECLARATION := '0' *)
IF rst OR set0 THEN
	q0 := NOT rst;
	q1 := q0;
	q2 := q0;
	q3 := q0;
	q4 := q0;
	q5 := q0;
	q6 := q0;
	q7 := q0;
ELSE
	IF D0 THEN Q0 := TRUE; END_IF;
	IF D1 THEN Q1 := TRUE; END_IF;
	IF D2 THEN Q2 := TRUE; END_IF;
	IF D3 THEN Q3 := TRUE; END_IF;
	IF D4 THEN Q4 := TRUE; END_IF;
	IF D5 THEN Q5 := TRUE; END_IF;
	IF D6 THEN Q6 := TRUE; END_IF;
	IF D7 THEN Q7 := TRUE; END_IF;

	IF clr AND NOT edge THEN
		IF q0 THEN q0 := FALSE;
		ELSIF q1 THEN q1 := FALSE;
		ELSIF q2 THEN q2 := FALSE;
		ELSIF q3 THEN q3 := FALSE;
		ELSIF q4 THEN q4 := FALSE;
		ELSIF q5 THEN q5 := FALSE;
		ELSIF q6 THEN q6 := FALSE;
		ELSE q7 := FALSE;
		END_IF;
	END_IF;
	edge := clr;
END_IF;

(* revision history
hm	25.12.2007	rev 1.0
	original version

hm	30. oct. 2008	rev 1.1
	optimized performance

hm	14. mar. 2009	rev 1.2
	removed double assignments

*)

END_FUNCTION_BLOCK

(* @NESTEDCOMMENTS := 'Yes' *)
(* @PATH := '\/Logic\/gate logic' *)
(* @OBJECTFLAGS := '0, 8' *)
(* @SYMFILEFLAGS := '2048' *)
FUNCTION BCDC_TO_INT : INT
VAR_INPUT
	IN : BYTE;
END_VAR

(*
version 1.1 30. jun. 2008
programmer 	hugo
tested by	oscat

this function converts a two digit bcd number into an integer.

*)

(* @END_DECLARATION := '0' *)
BCDC_TO_INT := (in AND 16#0F) + (SHR(in,4) * 10);

(* revision history
hm	13.12.2007	rev 1.0
	original version

hm	30.6.2008	rev 1.1
	changed name BCD_TO_INT to BCDC_TO_INT to avoid collision with util.lib

*)
END_FUNCTION

(* @NESTEDCOMMENTS := 'Yes' *)
(* @PATH := '\/Logic\/gate logic' *)
(* @OBJECTFLAGS := '0, 8' *)
(* @SYMFILEFLAGS := '2048' *)
FUNCTION BIT_COUNT : INT
VAR_INPUT
	IN : DWORD;
END_VAR

(*
version 1.1	10 sep 2007
programmer 	hugo
tested by		tobias

BIT_COUNT counts the amount True of bits in a dword.
for exabple: bit_count(3) returns 2 because two bits (bits 0 and 1) are true and all others are false.

*)
(* @END_DECLARATION := '0' *)
WHILE in > 0 DO
	IF in.0 THEN Bit_Count := Bit_Count + 1; END_IF;
	in := SHR(in,1);
END_WHILE;

(* revision history
5.7.2007	rev 1.0		original version

10.9.2007	rev 1.1		hm
	changed algorithm for better performace
	the execution time has reduced by a factor of 5
	deleted unused variable temp
*)
END_FUNCTION

(* @NESTEDCOMMENTS := 'Yes' *)
(* @PATH := '\/Logic\/gate logic' *)
(* @OBJECTFLAGS := '0, 8' *)
(* @SYMFILEFLAGS := '2048' *)
FUNCTION BIT_LOAD_B : BYTE
VAR_INPUT
	IN : BYTE;
	VAL : BOOL;
	POS : INT;
END_VAR
VAR CONSTANT
	dat : BYTE := 1;
END_VAR

(*
version 1.1	16. mar 2008
programmer 	hugo
tested by	tobias

this function loads a bit into a byte at position pos.
 *)
(* @END_DECLARATION := '0' *)
IF VAL THEN
	BIT_LOAD_B := in OR SHL(dat,pos);
ELSE
	BIT_LOAD_B := in AND (NOT SHL(dat,pos));
END_IF;

(* revision history
hm	29. feb 2008	rev 1.0
	original version

hm	16. mar 2008	rev 1.1
	change input bit to val for compatibility reasons
*)

END_FUNCTION

(* @NESTEDCOMMENTS := 'Yes' *)
(* @PATH := '\/Logic\/gate logic' *)
(* @OBJECTFLAGS := '0, 8' *)
(* @SYMFILEFLAGS := '2048' *)
FUNCTION BIT_LOAD_B2 : BYTE
VAR_INPUT
	I : BYTE;
	D : BOOL;
	P : INT;
	N : INT;
END_VAR

(*
version 1.0 18. oct. 2008
programmer 	hugo
tested by	tobias

this function loads N bits of D at pos P in Byte I

*)
(* @END_DECLARATION := '0' *)
IF D THEN
	BIT_LOAD_B2 := ROL(SHR(BYTE#255, 8 - N) OR ROR(i, P), P);
ELSE
	BIT_LOAD_B2 := ROL(SHL(BYTE#255, N) AND ROR(I, P), P);
END_IF;

(* revision history
hm	18. oct. 2008	rev 1.0
	original version

*)

END_FUNCTION

(* @NESTEDCOMMENTS := 'Yes' *)
(* @PATH := '\/Logic\/gate logic' *)
(* @OBJECTFLAGS := '0, 8' *)
(* @SYMFILEFLAGS := '2048' *)
FUNCTION BIT_LOAD_DW : DWORD
VAR_INPUT
	IN : DWORD;
	VAL : BOOL;
	POS : INT;
END_VAR
VAR CONSTANT
	dat : DWORD := 1;
END_VAR

(*
version 1.1	16. mar 2008
programmer 	hugo
tested by	tobias

this function loads a bit into a DWord at position pos.
 *)
(* @END_DECLARATION := '0' *)
IF val THEN
	BIT_LOAD_DW := in OR SHL(dat,pos);
ELSE
	BIT_LOAD_DW := in AND (NOT SHL(dat,pos));
END_IF;

(* revision history
hm	29. feb 2008	rev 1.0
	original version

hm	16. mar 2008	rev 1.1
	change input bit to val for compatibility reasons
*)

END_FUNCTION

(* @NESTEDCOMMENTS := 'Yes' *)
(* @PATH := '\/Logic\/gate logic' *)
(* @OBJECTFLAGS := '0, 8' *)
(* @SYMFILEFLAGS := '2048' *)
FUNCTION BIT_LOAD_DW2 : DWORD
VAR_INPUT
	I : DWORD;
	D : BOOL;
	P : INT;
	N : INT;
END_VAR

(*
version 1.0 18. oct. 2008
programmer 	hugo
tested by	tobias

this function loads N bits of D at pos P in DWORD I

*)
(* @END_DECLARATION := '0' *)
IF D THEN
	BIT_LOAD_DW2 := ROL(SHR(DWORD#4294967295, 32 - N) OR ROR(i, P), P);
ELSE
	BIT_LOAD_DW2 := ROL(SHL(DWORD#4294967295, N) AND ROR(I, P), P);
END_IF;

(* revision history
hm	18. oct. 2008	rev 1.0
	original version

*)

END_FUNCTION

(* @NESTEDCOMMENTS := 'Yes' *)
(* @PATH := '\/Logic\/gate logic' *)
(* @OBJECTFLAGS := '0, 8' *)
(* @SYMFILEFLAGS := '2048' *)
FUNCTION BIT_LOAD_W : WORD
VAR_INPUT
	IN : WORD;
	VAL : BOOL;
	POS : INT;
END_VAR
VAR CONSTANT
	dat : WORD := 1;
END_VAR

(*
version 1.1	16. mar 2008
programmer 	hugo
tested by	tobias

this function loads a bit into a Word at position pos.
 *)
(* @END_DECLARATION := '0' *)
IF val THEN
	BIT_LOAD_W := in OR SHL(dat,pos);
ELSE
	BIT_LOAD_W := in AND (NOT SHL(dat,pos));
END_IF;

(* revision history
hm	29. feb 2008	rev 1.0
	original version

hm	16. mar 2008	rev 1.1
	change input bit to val for compatibility reasons
*)

END_FUNCTION

(* @NESTEDCOMMENTS := 'Yes' *)
(* @PATH := '\/Logic\/gate logic' *)
(* @OBJECTFLAGS := '0, 8' *)
(* @SYMFILEFLAGS := '2048' *)
FUNCTION BIT_LOAD_W2 : WORD
VAR_INPUT
	I : WORD;
	D : BOOL;
	P : INT;
	N : INT;
END_VAR

(*
version 1.0 18. oct. 2008
programmer 	hugo
tested by	tobias

this function loads N bits of D at pos P in WORD I

*)
(* @END_DECLARATION := '0' *)
IF D THEN
	BIT_LOAD_W2 := ROL(SHR(WORD#65535, 16 - N) OR ROR(i, P), P);
ELSE
	BIT_LOAD_W2 := ROL(SHL(WORD#65535, N) AND ROR(I, P), P);
END_IF;

(* revision history
hm	18. oct. 2008	rev 1.0
	original version

*)

END_FUNCTION

(* @NESTEDCOMMENTS := 'Yes' *)
(* @PATH := '\/Logic\/gate logic' *)
(* @OBJECTFLAGS := '0, 8' *)
(* @SYMFILEFLAGS := '2048' *)
FUNCTION BIT_OF_DWORD : BOOL
VAR_INPUT
	in : DWORD;
	N : INT;
END_VAR

(*
version 1.2	6. jun. 2008
programmer 	hugo
tested by	tobias

this function extracts a single bit from the nth position from right (right is lowest bit)
the lowest Bit (Bit0 from in) is selected with N=0.
 *)
(* @END_DECLARATION := '0' *)
BIT_OF_DWORD := (SHR(in,N) AND 16#00000001) > 0;

(* old code used before rev 1.1
temp := SHR(in,n);
Bit_of_Dword := temp.0;
*)

(* revision history
hm	4. aug. 2006	rev 1.0
	original version

hm	29. feb 2008	rev 1.1
	improved performance

hm	6. jun. 2008	rev 1.2
	changes type of input N from byte to int
*)

END_FUNCTION

(* @NESTEDCOMMENTS := 'Yes' *)
(* @PATH := '\/Logic\/gate logic' *)
(* @OBJECTFLAGS := '0, 8' *)
(* @SYMFILEFLAGS := '2048' *)
FUNCTION BIT_TOGGLE_B : BYTE
VAR_INPUT
	IN : BYTE;
	POS : INT;
END_VAR

(*
version 1.0 18. oct. 2008
programmer 	hugo
tested by	tobias

this function toggles a bit of a BYTE at position pos.

*)
(* @END_DECLARATION := '0' *)
BIT_TOGGLE_B := SHL(BYTE#1, POS) XOR IN;

(* revision history
hm	18. oct. 2008	rev 1.0
	original version

*)

END_FUNCTION

(* @NESTEDCOMMENTS := 'Yes' *)
(* @PATH := '\/Logic\/gate logic' *)
(* @OBJECTFLAGS := '0, 8' *)
(* @SYMFILEFLAGS := '2048' *)
FUNCTION BIT_TOGGLE_DW : DWORD
VAR_INPUT
	IN : DWORD;
	POS : INT;
END_VAR

(*
version 1.0 18. oct. 2008
programmer 	hugo
tested by	tobias

this function toggles a bit of a WORD at position pos.

*)
(* @END_DECLARATION := '0' *)
BIT_TOGGLE_DW := SHL(DWORD#1, POS) XOR IN;

(* revision history
hm	18. oct. 2008	rev 1.0
	original version

*)

END_FUNCTION

(* @NESTEDCOMMENTS := 'Yes' *)
(* @PATH := '\/Logic\/gate logic' *)
(* @OBJECTFLAGS := '0, 8' *)
(* @SYMFILEFLAGS := '2048' *)
FUNCTION BIT_TOGGLE_W : WORD
VAR_INPUT
	IN : WORD;
	POS : INT;
END_VAR

(*
version 1.0 18. oct. 2008
programmer 	hugo
tested by	tobias

this function toggles a bit of a WORD at position pos.

*)
(* @END_DECLARATION := '0' *)
BIT_TOGGLE_W := SHL(WORD#1, POS) XOR IN;

(* revision history
hm	18. oct. 2008	rev 1.0
	original version

*)

END_FUNCTION

(* @NESTEDCOMMENTS := 'Yes' *)
(* @PATH := '\/Logic\/gate logic' *)
(* @OBJECTFLAGS := '0, 8' *)
(* @SYMFILEFLAGS := '2048' *)
FUNCTION BYTE_OF_BIT : BYTE
VAR_INPUT
	B0:BOOL;
	B1:BOOL;
	B2:BOOL;
	B3:BOOL;
	B4:BOOL;
	B5:BOOL;
	B6:BOOL;
	B7:BOOL;
END_VAR

(*
version 1.1	 18. feb 2006
programmer 	hugo
tested by		tobias

this function creates a byte from 8 individual bits

*)
(* @END_DECLARATION := '0' *)
Byte_of_bit := SHL(SHL(SHL(SHL(SHL(SHL(SHL(BOOL_TO_BYTE(B7),1) OR BOOL_TO_BYTE(B6),1) OR BOOL_TO_BYTE(B5),1) OR BOOL_TO_BYTE(B4),1)
	OR BOOL_TO_BYTE(B3),1) OR BOOL_TO_BYTE(B2),1) OR BOOL_TO_BYTE(B1),1) OR BOOL_TO_BYTE(B0);

(* revision history

hm	4. aug 2006		rev 1.0
	original version

hm	18. feb. 2008	rev 1.1
	improved performance

*)
END_FUNCTION

(* @NESTEDCOMMENTS := 'Yes' *)
(* @PATH := '\/Logic\/gate logic' *)
(* @OBJECTFLAGS := '0, 8' *)
(* @SYMFILEFLAGS := '2048' *)
FUNCTION BYTE_OF_DWORD : BYTE
VAR_INPUT
	in : DWORD;
	N : BYTE;
END_VAR

(*
version 1.2	30. oct. 2008
programmer 	hugo
tested by	oscat

this function extracts a single byte from the nth position from right (right is lowest byte)
the lower byte (starting with Bit0 from in) is selected with N=0.
*)

(* @END_DECLARATION := '0' *)
BYTE_OF_DWORD := DWORD_TO_BYTE(SHR(in,SHL(n,3)));

(* revision history
hm	17. jan 2007	rev 1.0
	original version

hm	2. jan 2008		rev 1.1
	improved performance

hm	30. oct. 2008	rev 1.2
	improved performance
*)

END_FUNCTION

(* @NESTEDCOMMENTS := 'Yes' *)
(* @PATH := '\/Logic\/gate logic' *)
(* @OBJECTFLAGS := '0, 8' *)
(* @SYMFILEFLAGS := '2048' *)
FUNCTION_BLOCK BYTE_TO_BITS
VAR_INPUT
	IN: BYTE;
END_VAR
VAR_OUTPUT
	B0: BOOL;
	B1: BOOL;
	B2: BOOL;
	B3: BOOL;
	B4: BOOL;
	B5: BOOL;
	B6: BOOL;
	B7: BOOL;
END_VAR

(*
version 1.1	16. mar. 2008
programmer 	hugo
tested by		tobias

this Function Block extracts the 8 Bits from a byte

*)
(* @END_DECLARATION := '0' *)
B0 := IN.0;
B1 := IN.1;
B2 := IN.2;
B3 := IN.3;
B4 := IN.4;
B5 := IN.5;
B6 := IN.6;
B7 := IN.7;

(* revision history
hm		4. aug 2006	rev 1.0
	original version

hm		16. mar 2008	rev 1.1
	renamed from byte_to_bit to byte_to_bits for compatibility reasons

*)
END_FUNCTION_BLOCK

(* @NESTEDCOMMENTS := 'Yes' *)
(* @PATH := '\/Logic\/gate logic' *)
(* @OBJECTFLAGS := '0, 8' *)
(* @SYMFILEFLAGS := '2048' *)
FUNCTION BYTE_TO_GRAY : BYTE
VAR_INPUT
	IN : BYTE;
END_VAR

(*
version 1.0	9. nov. 2009
programmer 	hugo
tested by		oscat

this function converts a binary to gray code

*)

(* @END_DECLARATION := '0' *)
BYTE_TO_GRAY := IN XOR SHR(IN,1);

(* revision history
hm	9. nov. 2009	rev 1.0
	original version

*)
END_FUNCTION

(* @NESTEDCOMMENTS := 'Yes' *)
(* @PATH := '\/Logic\/gate logic' *)
(* @OBJECTFLAGS := '0, 8' *)
(* @SYMFILEFLAGS := '2048' *)
FUNCTION CHECK_PARITY : BOOL
VAR_INPUT
	in : DWORD;
	p : BOOL;
END_VAR

(*
version 1.3	18 feb 2008
programmer 	hugo
tested by	tobias

this function checks for an even partity for a dword and partity bit.

*)
(* @END_DECLARATION := '0' *)
CHECK_PARITY := NOT p;
WHILE in > 0 DO
	CHECK_PARITY := CHECK_PARITY XOR in.0 XOR in.1 XOR in.2 XOR in.3;
	in := SHR(in,4);
END_WHILE;

(* code before rev 1.2
WHILE in > 0 DO
	IF in.0 THEN cnt := cnt + 1; END_IF;
	in := SHR(in,1);
END_WHILE;
check_parity := even(cnt) XOR P;
*)

(* revision history

rev 1.0 HM  1.oct.2006

rev 1.1 hm	10.sep.2007
	changed algorithm to improove performance

rev 1.2	hm	8 dec 2007
	changed algorithm to improove performance

rev 1.3 hm	18. feb 2008
	changed algorithm to improove performance
*)
END_FUNCTION

(* @NESTEDCOMMENTS := 'Yes' *)
(* @PATH := '\/Logic\/gate logic' *)
(* @OBJECTFLAGS := '0, 8' *)
(* @SYMFILEFLAGS := '2048' *)
FUNCTION CHK_REAL : BYTE
VAR_INPUT
	X : REAL;
END_VAR
VAR
	pt : REF_TO DWORD;
	tmp : DWORD;
END_VAR

(*
version 1.0	20. jan. 2011
programmer 	hugo
tested by		tobias

this function checks a floating point variable of type real (IEEE754-32Bits) for NAN and infinity
RETURN values: #0 = normal value, #20 = +infinity, #40 = -infinty, #80 = NAN

*)

(* @END_DECLARATION := '0' *)
pt := REF(X);				(* move real to dword, real_to_dword does not work becasze it treats dword as a number on many systems *)
tmp := ROL(pt^,1);			(* rotate left foir easy checking, sign will be at lease significant digit *)
IF tmp < 16#FF000000 THEN
	CHK_REAL := 16#00;		(* normalized and denormalized numbers *)
ELSIF tmp = 16#FF000000 THEN
	CHK_REAL := 16#20;		(* X is +infinity see IEEE754 *)
ELSIF tmp = 16#FF000001 THEN
	CHK_REAL := 16#40;		(* X is -infinity see IEEE754 *)
ELSE
	CHK_REAL := 16#80;		(* X is NAN see IEEE754 *)
END_IF;

(* revision history
hm	 20. jan. 2011	rev 1.0
	original version

*)
END_FUNCTION

(* @NESTEDCOMMENTS := 'Yes' *)
(* @PATH := '\/Logic\/gate logic' *)
(* @OBJECTFLAGS := '0, 8' *)
(* @SYMFILEFLAGS := '2048' *)
FUNCTION_BLOCK DEC_2
VAR_INPUT
	D: BOOL;
	A: BOOL;
END_VAR
VAR_OUTPUT
	Q0: BOOL;
	Q1: BOOL;
END_VAR

(*
version 1.1	3 Mar 2007
programmer 	hugo
tested by		tobias

a bit input will be decoded to the two outputs Q0 or Q1
dependent on the value of A
A=0 decodes to Q0 and A=1 decodes to Q1

*)
(* @END_DECLARATION := '0' *)
Q0 := D AND NOT A;
Q1 := D AND A;

(* revision history
hm 3.3.2007	rev 1.1
	rewritten in ST for better compatibility

*)
END_FUNCTION_BLOCK

(* @NESTEDCOMMENTS := 'Yes' *)
(* @PATH := '\/Logic\/gate logic' *)
(* @OBJECTFLAGS := '0, 8' *)
(* @SYMFILEFLAGS := '2048' *)
FUNCTION_BLOCK DEC_4
VAR_INPUT
	D: BOOL;
	A0: BOOL;
	A1: BOOL;
END_VAR
VAR_OUTPUT
	Q0: BOOL;
	Q1: BOOL;
	Q2: BOOL;
	Q3: BOOL;
END_VAR

(*
version 1.1	3 Mar 2007
programmer 	hugo
tested by		tobias

a bit input will be decoded to one of the 4 outputs
dependent on the Adress on A0 and A1

executioin TIME on wago 750-841 = 9us
*)
(* @END_DECLARATION := '0' *)
Q0 := D AND NOT A0 AND NOT A1;
Q1 := D AND A0 AND NOT A1;
Q2 := D AND NOT A0 AND A1;
Q3 := D AND A0 AND A1;

(* revision history
hm 3.3.2007	rev 1.1
	rewritten in ST for better compatibility

*)
END_FUNCTION_BLOCK

(* @NESTEDCOMMENTS := 'Yes' *)
(* @PATH := '\/Logic\/gate logic' *)
(* @OBJECTFLAGS := '0, 8' *)
(* @SYMFILEFLAGS := '2048' *)
FUNCTION_BLOCK DEC_8
VAR_INPUT
	D: BOOL;
	A0: BOOL;
	A1: BOOL;
	A2: BOOL;
END_VAR
VAR_OUTPUT
	Q0: BOOL;
	Q1: BOOL;
	Q2: BOOL;
	Q3: BOOL;
	Q4: BOOL;
	Q5: BOOL;
	Q6: BOOL;
	Q7: BOOL;
END_VAR
VAR
	X : INT;
END_VAR

(*
version 1.3	28. mar. 2009
programmer 	hugo
tested by		oscat

a bit input will be decoded to one of the 8 outputs
dependent on the Adress on A0, A1 and A2

*)
(* @END_DECLARATION := '0' *)
X.0 := A0; X.1 := A1; X.2 := A2;

Q0 := FALSE;
Q1 := FALSE;
Q2 := FALSE;
Q3 := FALSE;
Q4 := FALSE;
Q5 := FALSE;
Q6 := FALSE;
Q7 := FALSE;

CASE X OF
	0 : Q0 := D;
	1 : Q1 := D;
	2 : Q2 := D;
	3 : Q3 := D;
	4 : Q4 := D;
	5 : Q5 := D;
	6 : Q6 := D;
	7 : Q7 := D;
END_CASE;

(* revision history
hm 3. mar. 2007	rev 1.1
	rewritten in ST for better compatibility

hm	26. oct. 2008	rev 1.2
	code optimized

hm	28. mar. 2009	rev 1.3
	replaced multiple assignments
*)
END_FUNCTION_BLOCK

(* @NESTEDCOMMENTS := 'Yes' *)
(* @PATH := '\/Logic\/gate logic' *)
(* @OBJECTFLAGS := '0, 8' *)
(* @SYMFILEFLAGS := '2048' *)
FUNCTION DW_TO_REAL : REAL
VAR_INPUT
	X : DWORD;
END_VAR
VAR
	pt : REF_TO REAL;
END_VAR

(*
version 1.0	18. apr. 2008
programmer 	hugo
tested by		tobias

this function converts a DWORD to REAL in a bitwise manner.
*)

(* @END_DECLARATION := '0' *)
pt := REF(X);
DW_TO_REAL := pt^;

(* revision history
hm	18. apr. 2008
	original version

*)
END_FUNCTION

(* @NESTEDCOMMENTS := 'Yes' *)
(* @PATH := '\/Logic\/gate logic' *)
(* @OBJECTFLAGS := '0, 8' *)
(* @SYMFILEFLAGS := '2048' *)
FUNCTION DWORD_OF_BYTE : DWORD
VAR_INPUT
	B3 : BYTE;
	B2 : BYTE;
	B1 : BYTE;
	B0 : BYTE;
END_VAR

(*
version 1.3	18. jul. 2009
programmer 	hugo
tested by		tobias

this function creates a Dword from 4 individual bytes

*)
(* @END_DECLARATION := '0' *)
DWORD_OF_BYTE := SHL(SHL(SHL(BYTE_TO_DWORD(B3),8) OR BYTE_TO_DWORD(B2),8) OR BYTE_TO_DWORD(B1),8) OR BYTE_TO_DWORD(B0);

(* revision history
hm	24. jan 2007	rev 1.0
	original version

hm 2. jan 2008	rev 1.1
	inproved performance

hm	23. apr. 2008	rev 1.2
	reverse order of inputs to be more logical

hm	18. jul. 2009	rev 1.3
	added type conversions for compatibility reasons
*)
END_FUNCTION

(* @NESTEDCOMMENTS := 'Yes' *)
(* @PATH := '\/Logic\/gate logic' *)
(* @OBJECTFLAGS := '0, 8' *)
(* @SYMFILEFLAGS := '2048' *)
FUNCTION DWORD_OF_WORD : DWORD
VAR_INPUT
	W1 : WORD;
	W0 : WORD;
END_VAR

(*
version 1.0	18. jul. 2009
programmer 	hugo
tested by		tobias

this function creates a Dword from 2 individual Words

*)
(* @END_DECLARATION := '0' *)
DWORD_OF_WORD := SHL(WORD_TO_DWORD(W1),16) OR WORD_TO_DWORD(W0);

(* revision history

hm	18. jul. 2009	rev 1.0
	original version

*)
END_FUNCTION

(* @NESTEDCOMMENTS := 'Yes' *)
(* @PATH := '\/Logic\/gate logic' *)
(* @OBJECTFLAGS := '0, 8' *)
(* @SYMFILEFLAGS := '2048' *)
FUNCTION GRAY_TO_BYTE : BYTE
VAR_INPUT
	IN : BYTE;
END_VAR

(*
version 1.0	9. nov. 2009
programmer 	hugo
tested by		oscat

this function converts a gray code into binary

*)

(* @END_DECLARATION := '0' *)
GRAY_TO_BYTE := SHR(IN,4) XOR IN;
GRAY_TO_BYTE := SHR(GRAY_TO_BYTE,2) XOR GRAY_TO_BYTE;
GRAY_TO_BYTE := SHR(GRAY_TO_BYTE,1) XOR GRAY_TO_BYTE;

(* revision history
hm	9. nov. 2009	rev 1.0
	original version

*)
END_FUNCTION

(* @NESTEDCOMMENTS := 'Yes' *)
(* @PATH := '\/Logic\/gate logic' *)
(* @OBJECTFLAGS := '0, 8' *)
(* @SYMFILEFLAGS := '2048' *)
FUNCTION INT_TO_BCDC : BYTE
VAR_INPUT
	IN : INT;
END_VAR

(*
version 1.1	30. jun. 2008
programmer 	hugo
tested by		tobias

this function converts an integer into a two digit bcd number.
*)

(* @END_DECLARATION := '0' *)
INT_TO_BCDC := SHL(INT_TO_BYTE(IN / INT#10),4) OR INT_TO_BYTE(in MOD INT#10);

(* revision history
hm	13.12.2007
	original version

hm	30.6.2008	rev 1.1
	changed name INT_TO_BCD to INT_TO_BCDC to avoid collision with util.lib
	corrected error in code

*)
END_FUNCTION

(* @NESTEDCOMMENTS := 'Yes' *)
(* @PATH := '\/Logic\/gate logic' *)
(* @OBJECTFLAGS := '0, 8' *)
(* @SYMFILEFLAGS := '2048' *)
FUNCTION MUX_2 : BOOL
VAR_INPUT
	D0: BOOL;
	D1: BOOL;
	A0: BOOL;
END_VAR

(*
	version 1.2	16. oct. 2008
	programmer 	hugo
	tested BY	oscat

	dual input multiplexer
	depending on the value of A0, D0 or D1 will be switched to the Output

	executioin TIME on wago 750-841 = 7us
*)
(* @END_DECLARATION := '0' *)
MUX_2 := SEL(A0, D0, D1);

(*
revision history:
hm	5.10.2006		rev 1.1
	changed to ST Langage for better portability.

hm	16. oct. 2008	rev 1.2
	improved performance

*)
END_FUNCTION

(* @NESTEDCOMMENTS := 'Yes' *)
(* @PATH := '\/Logic\/gate logic' *)
(* @OBJECTFLAGS := '0, 8' *)
(* @SYMFILEFLAGS := '2048' *)
FUNCTION MUX_4 : BOOL
VAR_INPUT
	D0: BOOL;
	D1: BOOL;
	D2: BOOL;
	D3: BOOL;
	A0: BOOL;
	A1: BOOL;
END_VAR

(*
version 1.2	16. oct. 2008
programmer 	hugo
tested BY	oscat

quad input multiplexer
depending on the value of A0 and A1, one of the 4 inputs will be switched to the Output

*)
(* @END_DECLARATION := '0' *)
IF A1 THEN
	MUX_4 := SEL(A0, D2, D3);
ELSE
	MUX_4 := SEL(A0, D0, D1);
END_IF;

(*
revision history:
hm 	5.10.2006		rev 1.1
	rewritten to ST for better portability

hm	16. oct. 2008	rev 1.2
	improved performance

*)
END_FUNCTION

(* @NESTEDCOMMENTS := 'Yes' *)
(* @PATH := '\/Logic\/gate logic' *)
(* @OBJECTFLAGS := '0, 8' *)
(* @SYMFILEFLAGS := '2048' *)
FUNCTION PARITY : BOOL
VAR_INPUT
	in : DWORD;
END_VAR

(*
	version 1.3	18 feb 2008
	programmer 	hugo
	tested BY		hans

this function calculates the even parity of an input Dword
the output will be true if the amount of high bits are an odd number.

*)

(* @END_DECLARATION := '0' *)
WHILE in > 0 DO
	PARITY := PARITY XOR in.0 XOR in.1 XOR in.2 XOR in.3;
	in := SHR(in,4);
END_WHILE;

(* code before rev 1.2
WHILE in > 0 DO
	IF in.0 THEN cnt := cnt +1; END_IF;
	in := SHR(in,1);
END_WHILE;
IF (cnt MOD 2) = 1 THEN parity := TRUE; ELSE parity := FALSE; END_IF;
*)

(* revision history

rev 1.0 hm 1 sep 2006
	original version

rev 1.1 hm 10.9.2007
	changed algorithm to improve performance

rev 1.2	hm	8 dec 2007
	changed algorithm to improve performance

rev 1.3	hm	18 feb 2008
	changed algorithm to improve performance
*)
END_FUNCTION

(* @NESTEDCOMMENTS := 'Yes' *)
(* @PATH := '\/Logic\/gate logic' *)
(* @OBJECTFLAGS := '0, 8' *)
(* @SYMFILEFLAGS := '2048' *)
FUNCTION REAL_TO_DW : DWORD
VAR_INPUT
	X : REAL;
END_VAR
VAR
	pt : REF_TO DWORD;
END_VAR

(*
version 1.0	18. apr. 2008
programmer 	hugo
tested by		tobias

this function converts a 32 Bit Real to a dword in a bitwise manner.
*)

(* @END_DECLARATION := '0' *)
pt := REF(X);
REAL_TO_DW := pt^;

(* revision history
hm	18. apr. 2008
	original version

*)
END_FUNCTION

(* @NESTEDCOMMENTS := 'Yes' *)
(* @PATH := '\/Logic\/gate logic' *)
(* @OBJECTFLAGS := '0, 8' *)
(* @SYMFILEFLAGS := '2048' *)
FUNCTION REFLECT : DWORD
VAR_INPUT
	D : DWORD;
	L : INT;
END_VAR
VAR
	i : INT;
END_VAR

(*
	version 1.0	16. jan 2011
	programmer 	hugo
	tested BY		tobias

This function reverses the specified amount of bits from bit 0 to bit n within a dword  while L specifies the amount of Bits to be reflected.

*)

(* @END_DECLARATION := '0' *)
REFLECT := 0;
FOR i := 1 TO L DO
	REFLECT := SHL(REFLECT, 1) OR BOOL_TO_DWORD(D.0);
	D := SHR(D, 1);
END_FOR;
REFLECT := REFLECT OR SHL(D, L);

(* revision history
hm	 16. jan 2011
	new module

*)
END_FUNCTION

(* @NESTEDCOMMENTS := 'Yes' *)
(* @PATH := '\/Logic\/gate logic' *)
(* @OBJECTFLAGS := '0, 8' *)
(* @SYMFILEFLAGS := '2048' *)
FUNCTION REVERSE : BYTE
VAR_INPUT
	IN : BYTE;
END_VAR

(*
	version 1.1	18. feb 2008
	programmer 	hugo
	tested BY		tobias

This function reverses the bits of a byte so that after execution bit 7 is at bit 0 location and so forth.

*)
(* @END_DECLARATION := '0' *)
REVERSE := SHL(in,7) OR SHR(in,7) OR (ROR(in,3) AND 2#01000100) OR (ROL(in,3) AND 2#00100010)
	OR (SHL(in,1) AND 2#00010000) OR (SHR(in,1) AND 2#00001000);

(* revision history
hm		9.oct 2007		rev 1.0
	original version

hm		18. feb 2008	rev 1.1
	improved performance
*)
END_FUNCTION

(* @NESTEDCOMMENTS := 'Yes' *)
(* @PATH := '\/Logic\/gate logic' *)
(* @OBJECTFLAGS := '0, 8' *)
(* @SYMFILEFLAGS := '2048' *)
FUNCTION SHL1 : DWORD
VAR_INPUT
	IN : DWORD;
	N : INT;
END_VAR
VAR CONSTANT
	temp : DWORD := 16#FFFF_FFFF;
END_VAR

(*
version 1.1	27 dec 2007
programmer 	hugo
tested by		tobias

SHL1 shifts N bits to the left filling the new bits with 1

*)
(* @END_DECLARATION := '0' *)
SHL1 := SHR(temp,32-N) OR SHL(IN,N);

(* revision history
hm	14.9.2007		rev 1.0
	original version

hm	27. dec 2007	rev 1.1
	changed code for better performance

*)
END_FUNCTION

(* @NESTEDCOMMENTS := 'Yes' *)
(* @PATH := '\/Logic\/gate logic' *)
(* @OBJECTFLAGS := '0, 8' *)
(* @SYMFILEFLAGS := '2048' *)
FUNCTION SHR1 : DWORD
VAR_INPUT
	IN : DWORD;
	N : INT;
END_VAR
VAR CONSTANT
	temp : DWORD := 16#FFFF_FFFF;
END_VAR

(*
version 1.1	27 dec 2007
programmer 	hugo
tested by		tobias

SHR1 shifts N bits to the right filling the new bits with 1

*)
(* @END_DECLARATION := '0' *)
SHR1 := SHL(temp,32-N) OR SHR(IN,N);

(* revision history
hm	14.9.2007		rev 1.0
	original version

hm	27. dec 2007	rev 1.1
	changed code for better performance

*)
END_FUNCTION

(* @NESTEDCOMMENTS := 'Yes' *)
(* @PATH := '\/Logic\/gate logic' *)
(* @OBJECTFLAGS := '0, 8' *)
(* @SYMFILEFLAGS := '2048' *)
FUNCTION SWAP_BYTE : WORD
VAR_INPUT
	IN : WORD;
END_VAR

(*
version 1.0	4 feb 2008
programmer 	hugo
tested by		tobias

This function swaps the high and low byte of the word in.

*)
(* @END_DECLARATION := '0' *)
SWAP_BYTE := ROL(in,8);

(* revision history
hm		4. feb 2008	rev 1.0
	original version

*)
END_FUNCTION

(* @NESTEDCOMMENTS := 'Yes' *)
(* @PATH := '\/Logic\/gate logic' *)
(* @OBJECTFLAGS := '0, 8' *)
(* @SYMFILEFLAGS := '2048' *)
FUNCTION SWAP_BYTE2 : DWORD
VAR_INPUT
	IN : DWORD;
END_VAR

(*
version 1.0	4 feb 2008
programmer 	hugo
tested by		tobias

This function reverses the byte order in the dword.

*)
(* @END_DECLARATION := '0' *)
Swap_Byte2 := (ROR(in,8) AND 16#FF00FF00) OR (ROL(in,8) AND 16#00FF00FF);

(* revision history
hm		4. feb 2008	rev 1.0
	original version

*)

END_FUNCTION

(* @NESTEDCOMMENTS := 'Yes' *)
(* @PATH := '\/Logic\/gate logic' *)
(* @OBJECTFLAGS := '0, 8' *)
(* @SYMFILEFLAGS := '2048' *)
FUNCTION WORD_OF_BYTE : WORD
VAR_INPUT
	B1 : BYTE;
	B0 : BYTE;
END_VAR

(*
version 1.4	18. jul. 2009
programmer 	hugo
tested by		tobias

this function creates a word from 2 individual bytes

*)
(* @END_DECLARATION := '0' *)
WORD_OF_BYTE := SHL(BYTE_TO_WORD(B1),8) OR BYTE_TO_WORD(B0);

(* revision history
hm	24. jan 2007	rev 1.0
	original version

hm	2. jan 2008	rev 1.1
	improved performance

hm	19. feb 2008	rev 1.2
	replaced and with or for better compatibility

hm	23. apr. 2008	rev 1.3
	reverse order of inputs to be more logical

hm	18. jul. 2009	rev 1.4
	added type conversions for compatibility reasons

*)
END_FUNCTION

(* @NESTEDCOMMENTS := 'Yes' *)
(* @PATH := '\/Logic\/gate logic' *)
(* @OBJECTFLAGS := '0, 8' *)
(* @SYMFILEFLAGS := '2048' *)
FUNCTION WORD_OF_DWORD : WORD
VAR_INPUT
	in : DWORD;
	N : BYTE;
END_VAR

(*
version 1.2	30. oct. 2008
programmer 	hugo
tested by	oscat

this function extracts a single word from the nth position from right (right is lowest byte)
the lower word (starting with Bit0 from in) is selected with N=0.
*)

(* @END_DECLARATION := '0' *)
WORD_OF_DWORD := DWORD_TO_WORD(SHR(in,SHL(n,4)));

(* revision history
hm	17. jan 2007	rev 1.0
	original version

hm	2. jan 2008		rev 1.1
	improved performance

hm	30. oct. 2008	rev 1.2
	improved performance
*)

END_FUNCTION

(* @NESTEDCOMMENTS := 'Yes' *)
(* @PATH := '\/Logic\/generators' *)
(* @OBJECTFLAGS := '0, 8' *)
(* @SYMFILEFLAGS := '2048' *)
FUNCTION_BLOCK A_TRIG
VAR_INPUT
	IN : REAL;
	RES : REAL;
END_VAR
VAR_OUTPUT
	Q : BOOL;
	D : REAL;
END_VAR
VAR
	last_in : REAL;
END_VAR

(*
version 1.1	25. oct. 2008
programmer 	hugo
tested by	oscat

this block is similar to the IEC Standard R_trig and F_trig but it monitors a REAL for change.
if the valiue on IN changes more then D from the last value it will generate trigger and display the difference in output D.
the trigger will only be active for one cycle.

*)

(* @END_DECLARATION := '0' *)
D := IN - LAST_IN;
Q := ABS(D) > res;
IF Q THEN last_in := IN; END_IF;
D := IN - LAST_IN;

(* revision history

hm 	16. jul. 2008	rev 1.0
	original version released

hm	25. oct. 2008	rev 1.1
	code optimization
	a_trig now also works for res = 0

*)
END_FUNCTION_BLOCK

(* @NESTEDCOMMENTS := 'Yes' *)
(* @PATH := '\/Logic\/generators' *)
(* @OBJECTFLAGS := '0, 8' *)
(* @SYMFILEFLAGS := '2048' *)
FUNCTION_BLOCK B_TRIG
VAR_INPUT
	CLK : BOOL;
END_VAR
VAR_OUTPUT
	Q : BOOL;
END_VAR
VAR
	edge : BOOL;
END_VAR

(*
version 1.0	4. aug. 2006
programmer 	hugo
tested by		tobias

this block is similar to R_trig and F_trig but it generates a pulse on rising and falling edge.

*)

(* @END_DECLARATION := '0' *)
Q := clk XOR edge;
edge := CLK;

(* revision history
hm		4. aug. 2006	rev 1.0
	original version

*)
END_FUNCTION_BLOCK

(* @NESTEDCOMMENTS := 'Yes' *)
(* @PATH := '\/Logic\/generators' *)
(* @OBJECTFLAGS := '0, 8' *)
(* @SYMFILEFLAGS := '2048' *)
FUNCTION_BLOCK CLICK_CNT
VAR_INPUT
	IN : BOOL;
	N : INT;
	TC : TIME;
END_VAR
VAR_OUTPUT
	Q : BOOL;
END_VAR
VAR
	tx : TP;
	edge: BOOL;
	cnt: INT := -1;
END_VAR

(*
version 1.0	16. jul. 2008
programmer 	hugo
tested by	oscat

this Module decodes a specified number of clicks.
the output trig is high for one cycle if N clicks are present within a specified time TC.

*)

(* @END_DECLARATION := '0' *)
(* Q shall only be active for one cycle only *)
Q := FALSE;

IF in AND NOT edge AND NOT tx.q THEN
	(* a rising edge on in sets the counter to 0 *)
	cnt := 0;
ELSIF tx.Q AND NOT IN AND edge THEN
	(* count falling edges when tp.q is true *)
	cnt := cnt + 1;
ELSIF NOT tx.Q THEN
	Q := cnt = N;
	cnt := -1;
END_IF;

(* remember the status of IN *)
edge := IN;
tx(in := IN, pt := TC);

(* revision history

hm 	16. jul. 2008	rev 1.0
	original version released

*)
END_FUNCTION_BLOCK

(* @NESTEDCOMMENTS := 'Yes' *)
(* @PATH := '\/Logic\/generators' *)
(* @OBJECTFLAGS := '0, 8' *)
(* @SYMFILEFLAGS := '2048' *)
FUNCTION_BLOCK CLICK_DEC
VAR_INPUT
	IN : BOOL;
	TC : TIME;
END_VAR
VAR_OUTPUT
	Q0, Q1, Q2, Q3 : BOOL;
END_VAR
VAR
	tx : TP;
	edge: BOOL;
	cnt: INT := -1;
END_VAR

(*
version 1.1	14. mar. 2009
programmer 	hugo
tested by		oscat

this Module detects a rising edge on In and decodes the amount of falling edges (Pulses) within a specified time TC.
the outputs Q0..Q3 will go true for one cycle and the amount of clicks within a specified time TC.
if only a rising egde is detected within TC Q0 will respond, Q1 for 1 pulse and so on..

*)

(* @END_DECLARATION := '0' *)
(* Q shall only be active for one cycle only *)
IF in = FALSE THEN
	Q0 := FALSE;
	Q1 := FALSE;
	Q2:= FALSE;
	Q3 := FALSE;
END_IF;

IF in AND NOT edge AND NOT tx.q THEN
	(* a rising edge on in sets the counter to 0 *)
	cnt := 0;
ELSIF tx.Q AND NOT IN AND edge THEN
	(* count falling edges when tp.q is true *)
	cnt := cnt + 1;
ELSIF NOT tx.Q THEN
	CASE cnt OF
		0 : Q0 := TRUE;
		1 : Q1 := TRUE;
		2 : Q2 := TRUE;
		3 : Q3 := TRUE;
	END_CASE;
	cnt := -1;
END_IF;

(* remember the status of IN *)
edge := IN;
tx(in := IN, pt := TC);

(* revision history

hm 17. jul. 2008	rev 1.0
	original version released

hm	14. mar. 2009	rev 1.1
	removed double assignments

*)
END_FUNCTION_BLOCK

(* @NESTEDCOMMENTS := 'Yes' *)
(* @PATH := '\/Logic\/generators' *)
(* @OBJECTFLAGS := '0, 8' *)
(* @SYMFILEFLAGS := '2048' *)
FUNCTION_BLOCK CLK_DIV
VAR_INPUT
	clk : BOOL;
	rst: BOOL;
END_VAR
VAR_OUTPUT
	Q0 : BOOL;
	Q1 : BOOL;
	Q2 : BOOL;
	Q3 : BOOL;
	Q4 : BOOL;
	Q5 : BOOL;
	Q6 : BOOL;
	Q7 : BOOL;
END_VAR
VAR
	cnt: BYTE;
END_VAR

(*
version 1.1	2 jan 2008
programmer 	hugo
tested by		tobias

this is a clock divider
each output divides the signal by 2
Q0 = clk / 2 , Q1 = Q0 / 2 and so on.
the outputs have a 50% duty cycle each.

*)

(* @END_DECLARATION := '0' *)
IF rst THEN
	cnt:= 0;
	Q0 := 0;
	Q1 := 0;
	Q2 := 0;
	Q3 := 0;
	Q4 := 0;
	Q5 := 0;
	Q6 := 0;
	Q7 := 0;
ELSIF clk THEN
	cnt:= cnt +1;
	Q0 := cnt.0;
	Q1 := cnt.1;
	Q2 := cnt.2;
	Q3 := cnt.3;
	Q4 := cnt.4;
	Q5 := cnt.5;
	Q6 := cnt.6;
	Q7 := cnt.7;
END_IF;

(* revision history
hm	4. aug. 2006	rev 1.0
	original version

hm	2. jan 2008		rev 1.1
	improved performance

*)
END_FUNCTION_BLOCK

(* @NESTEDCOMMENTS := 'Yes' *)
(* @PATH := '\/Logic\/generators' *)
(* @OBJECTFLAGS := '0, 8' *)
(* @SYMFILEFLAGS := '2048' *)
FUNCTION_BLOCK CLK_N
VAR_INPUT
	N : INT;
END_VAR
VAR_OUTPUT
	Q : BOOL;
END_VAR
VAR
	edge : BOOL;
	stime: DWORD;
	clk: BOOL;
END_VAR

(*
version 1.0	17 sep 2007
programmer 	hugo
tested by		tobias

clk_N uses the internal sps time to generate one pulse every N ms
every pulse is only valid for one cycle so that a edge trigger is not necessary
clk_N generates pulses depending on the accuracy of the system clock.
The input N controlls the period time of the clock.
N=0 equals 1ms, N=1 equals 2ms, N=2 equals 4ms, N=3 equals 8ms ....

be careful, 1ms clocks will only work on very powerful sps cpu's
*)
(* @END_DECLARATION := '0' *)
stime := SHR(T_PLC_MS(),N);
clk := stime.0;
Q := clk XOR edge;
edge := CLK;

(* revision history
hm	16. dec 2007		rev 1.0
	original version

*)
END_FUNCTION_BLOCK

(* @NESTEDCOMMENTS := 'Yes' *)
(* @PATH := '\/Logic\/generators' *)
(* @OBJECTFLAGS := '0, 8' *)
(* @SYMFILEFLAGS := '2048' *)
	FUNCTION_BLOCK CLK_PRG
VAR_INPUT
	PT : TIME := t#10ms;
END_VAR
VAR_OUTPUT
	Q : BOOL;
END_VAR
VAR
	init : BOOL;
	last : TIME;
	tx: TIME;
END_VAR

(*
version 1.3	25. oct. 2008
programmer 	hugo
tested by		tobias

clk_prg uses the internal sps time to generate a clock with programmable period time.
the first cycle after start is a clk pulse and then depending on the programmed period time a delay.
every pulse is only valid for one cycle.
the accuracy of clk_prg is depending on the accuracy of the system clock.

*)
(* @END_DECLARATION := '0' *)
(* read system time *)
tx := DWORD_TO_TIME(T_PLC_MS());

(* initialize on startup *)
IF NOT init THEN
	init := TRUE;
	last := tx - pt;
END_IF;

(* generate output pulse when next_pulse is reached *)
Q := tx - last >= pt;
IF Q THEN last := tx; END_IF;

(* revision hiostory

hm 25 feb 2007	rev 1.1
	rewritten code for higher performance
	pt can now be changed during runtime

hm	17. sep 2007	rev 1.2
	replaced time() with t_plc_ms() for compatibility reasons

hm	25. oct. 2008	rev 1.3
	optimized code

*)
END_FUNCTION_BLOCK

(* @NESTEDCOMMENTS := 'Yes' *)
(* @PATH := '\/Logic\/generators' *)
(* @OBJECTFLAGS := '0, 8' *)
(* @SYMFILEFLAGS := '2048' *)
FUNCTION_BLOCK CLK_PULSE
VAR_INPUT
	PT : TIME;
	N : INT;
	RST : BOOL ;
END_VAR
VAR_OUTPUT
	Q : BOOL;
	CNT : INT;
	RUN : BOOL;
END_VAR
VAR
	tx, tn: DWORD;
	init: BOOL;
END_VAR

(*
version 1.2		16 feb 2011
programmer 	hugo
tested by		oscat

clk_pulse uses the internal sps time to generate a clock with programmable period time.
the period time is defined for 10ms .. 65s.
pulse generation is continuous if N = 0 and for n pulses otherwise.
the first cycle after start is a clk pulse and then depending on the programmed period time a delay.
every pulse is only valid for one cycle so that a edge trigger is not necessary
clk_prg depending on the accuracy of the system clock.

*)
(* @END_DECLARATION := '0' *)
tx := T_PLC_MS();		(* read system *)
Q := FALSE;				(* reset Q we generate pulses only for one cycle *)
RUN := CNT < N;

IF NOT init OR RST THEN
	init := TRUE;
	CNT := 0;
	tn := tx - TIME_TO_DWORD(PT);
	RUN := FALSE;
ELSIF (cnt < N OR N = 0) AND tx - tn >= TIME_TO_DWORD(PT) THEN		(* generate a pulse *)
	CNT := CNT + 1;
	Q := TRUE;
	tn := tn + TIME_TO_DWORD(PT);
END_IF;

(* revision history
hm		4. aug 2006		rev 1.0
	original version

hm		17. sep 2007	rev 1.1
	replaced time() with T_PLC_S() for compatblity reasons

hm		16. feb. 2011	rev 1.2
	fixed an error when timer overflows
*)
END_FUNCTION_BLOCK

(* @NESTEDCOMMENTS := 'Yes' *)
(* @PATH := '\/Logic\/generators' *)
(* @OBJECTFLAGS := '0, 8' *)
(* @SYMFILEFLAGS := '2048' *)
FUNCTION_BLOCK CYCLE_4
VAR_INPUT
	E : BOOL := TRUE;
	T0, T1, T2, T3 : TIME;
	S0 : BOOL;
	SX : INT;
	SL : BOOL;
END_VAR
VAR_OUTPUT
	STATE : INT;
END_VAR
VAR
	tx : TIME;
	last : TIME;
	init: BOOL;
END_VAR

(*
version 1.0
programmer 	hugo
tested by	oscat

*)
(* @END_DECLARATION := '0' *)
(* read system timer *)
tx := DWORD_TO_TIME(T_PLC_MS());
(* init on first cycle *)
IF NOT init THEN
	init := TRUE;
	last := tx;
END_IF;

IF E THEN
	IF SL THEN
		(* when sx > 0 then the state sx is forced to start *)
		state:= LIMIT(0,SX,3);
		last := tx;
		(* this is to avoid to reset sx from the calling programm it does work fine on codesys but i am not sure about other systems, because we are writing to an input *)
		SL := FALSE;
	ELSE
		CASE state OF
			0 :	(* wait for T0 and switch to next cycle *)
				IF tx - last >= T0 THEN
					state := 1;
					last := tx;
				END_IF;
			1 : (* wait for T1 over 1st cycle *)
				IF tx - last >= T1 THEN
					state := 2;
					last := tx;
				END_IF;
			2 : (* wait for T1 over 1st cycle *)
				IF tx - last >= T2 THEN
					state := 3;
					last := tx;
				END_IF;
			3 : (* wait for T2 over 2nd cycle *)
				IF tx - last >= T3 THEN
					IF S0 THEN State := 0; END_IF; (* if S0 is false, the sequence stops at state 3 *)
					last := tx;
				END_IF;
		END_CASE;
	END_IF;
ELSE
	state := 0;
	last := tx;
END_IF;

(*
hm	3. nov. 2008	rev 1.0
	original version

*)
END_FUNCTION_BLOCK

(* @NESTEDCOMMENTS := 'Yes' *)
(* @PATH := '\/Logic\/generators' *)
(* @OBJECTFLAGS := '0, 8' *)
(* @SYMFILEFLAGS := '2048' *)
FUNCTION_BLOCK D_TRIG
VAR_INPUT
	in : DWORD;
END_VAR
VAR_OUTPUT
	Q : BOOL;
	X : DWORD;
END_VAR
VAR
	last_in : DWORD;
END_VAR

(*
version 1.1	19. feb 2008
programmer 	hugo
tested by		tobias

this block is similar to the IEC Standard R_trig and F_trig but it monitors a DWORD, WORD or Byte Variable instead and generated an Output Pulse for one cycle only when the input has changed.
an additional output x (Dword) will state the chage of the input.
Example: the input has chaged from 0001 to 0010 then the output x will be 2.

*)

(* @END_DECLARATION := '0' *)
Q := in <> last_in;
X := in - last_in;
last_in := in;

(* revision history

hm 	4.09.2007		rev 1.0
	original version released

hm	19. feb. 2008	rev 1.1
	performance improvement
*)
END_FUNCTION_BLOCK

(* @NESTEDCOMMENTS := 'Yes' *)
(* @PATH := '\/Logic\/generators' *)
(* @OBJECTFLAGS := '0, 8' *)
(* @SYMFILEFLAGS := '2048' *)
FUNCTION_BLOCK GEN_BIT
VAR_INPUT
	in0 : DWORD;
	in1 : DWORD;
	in2 : DWORD;
	in3 : DWORD;
	clk : BOOL;
	steps : INT;
	rep : INT;
	rst : BOOL;
END_VAR
VAR_OUTPUT
	Q0 :BOOL;
	Q1 :BOOL;
	Q2 :BOOL;
	Q3 :BOOL;
	cnt : INT;
	run : BOOL;
END_VAR
VAR
	r0: DWORD;
	r1: DWORD;
	r2: DWORD;
	r3: DWORD;
	rx : INT := 1;
END_VAR

(*
version 1.2	14. mar. 2009
programmer 	hugo
tested by		tobias

gen_bit is 4 bit sequencial pattern generator with 4 DWORD inputs and 4 serial outputs.
with the first clock pulse after a reset or after power on, bit 0 of the input DWORDS IN is present on the Outputs Q and the next clock cycle shifts to Bit 1 and so on.
the input steps defines how many bits of the input dwords will be shifted to the outputs. the sequence can be repetive when rep = 0 or any amount of repetitions can be defined with input rep.

*)
(* @END_DECLARATION := '0' *)
(* check if number of runs is finished or rep = 0 which means continuous *)

IF clk AND NOT rst THEN
	run := (rep = 0) OR (rx <= rep);
	IF run THEN
		(* check for step counter reached and reset to 0 if cnt = steps *)
		IF cnt = steps THEN
			cnt := 0;
		END_IF;

		(* when cnt = 0 then reload the inputs into the registers *)
		IF cnt = 0 THEN
			r0 := in0;
			r1 := in1;
			r2 := in2;
			r3 := in3;
		END_IF;

		(* when cnt < steps, shift the lowest bits to the outputs *)
		IF (cnt < steps) THEN
			Q0 := r0.0;
			Q1 := r1.0;
			Q2 := r2.0;
			Q3 := r3.0;
			r0 := SHR(r0,1);
			r1 := SHR(r1,1);
			r2 := SHR(r2,1);
			r3 := SHR(r3,1);
		END_IF;

		(* increment the step counter *)
		cnt := cnt +1;
		IF (cnt = steps) AND (rep <> 0) THEN rx := rx +1; END_IF;
		IF (rx > rep) AND (rep <> 0) THEN run := FALSE; END_IF;
	END_IF;
ELSE
	IF rst THEN
		run := FALSE;
		Q0 := FALSE;
		Q1 := FALSE;
		Q2 := FALSE;
		Q3 := FALSE;
		r0 := 0;
		r1 := 0;
		r2 := 0;
		r3 := 0;
		cnt := 0;
		rx := 1;
	END_IF;
END_IF;

(* revision histroy
hm	4 aug 2006	rev 1.0
	original version

hm 15. oct. 2008	rev 1.1
	improved performance

hm	14. mar. 2009	rev 1.2
	removed double assignments

*)
END_FUNCTION_BLOCK

(* @NESTEDCOMMENTS := 'Yes' *)
(* @PATH := '\/Logic\/generators' *)
(* @OBJECTFLAGS := '0, 8' *)
(* @SYMFILEFLAGS := '2048' *)
FUNCTION_BLOCK GEN_SQ
VAR_INPUT
	PT : TIME;
END_VAR
VAR_OUTPUT
	Q : BOOL;
END_VAR
VAR
	tn: DWORD;
	tx: DWORD;
	init : BOOL;
END_VAR

(*
version 1.3	16. feb. 2011
programmer 	hugo
tested by		tobias

gen_sq generates square wave signal with programmable period time.

*)
(* @END_DECLARATION := '0' *)
(* read system time *)
tx := T_PLC_MS();

IF NOT init THEN
	init := TRUE;
	tn := tx;
	Q := TRUE;
ELSIF tx - tn >= SHR(TIME_TO_DWORD(PT),1) THEN
	Q := NOT Q;
	tn := tn + SHR(TIME_TO_DWORD(pt),1);
END_IF;

(* revision history
hm	4. aug 2006	rev 1.0
	original version

hm	17. sep 2007	rev 1.1
	replaced time() with T_PLC_MS() for compatibility reasons

hm	18. jul. 2009	rev 1.2
	improved accuracy

hm	16. feb 2011	rev 1.3
	corrected an error with timer overflow
*)

END_FUNCTION_BLOCK

(* @NESTEDCOMMENTS := 'Yes' *)
(* @PATH := '\/Logic\/generators' *)
(* @OBJECTFLAGS := '0, 8' *)
(* @SYMFILEFLAGS := '2048' *)
FUNCTION_BLOCK SCHEDULER
VAR_INPUT
	E0 : BOOL;
	E1 : BOOL;
	E2 : BOOL;
	E3 : BOOL;
END_VAR
VAR_INPUT (* CONSTANT *)
	T0, T1, T2, T3 : TIME;
END_VAR
VAR_OUTPUT
	Q0, Q1, Q2, Q3 : BOOL;
END_VAR
VAR
	init : BOOL;
	s0, s1, s2, s3 : TIME;
	tx : TIME;
	c : INT;
END_VAR

(*
version 1.1	14. mar. 2009
programmer 	hugo
tested by		tobias

SCHEDULER is used to call programs or function blocks at specific intervals.
T0..T3 defines the interval times.

*)

(* @END_DECLARATION := '0' *)
(* read system_time *)
tx := DWORD_TO_TIME(T_PLC_MS());

IF NOT init THEN
	init := TRUE;
	s0 := tx - T0;
	s1 := tx - T1;
	s2 := tx - T2;
	s3 := tx - T3;
END_IF;

Q0 := FALSE;
Q1 := FALSE;
Q2 := FALSE;
Q3 :=FALSE;

CASE c OF
	0: 	IF tx - s0 >= T0 THEN
			Q0 := E0;
			s0 := tx;
		END_IF;
		c := 1;
	1: 	IF tx - s1 >= T1 THEN
			Q1 := E1;
			s1 := tx;
		END_IF;
		c := 2;
	2: 	IF tx - s2 >= T2 THEN
			Q2 := E2;
			s2 := tx;
		END_IF;
		c := 3;
	3: 	IF tx - s3 >= T3 THEN
			Q3 := E3;
			s3 := tx;
		END_IF;
		c := 0;
END_CASE;

(* revision history

hm 28. sep. 2008	rev 1.0
	original version

hm	14. mar. 2009	rev 1.1
	removed double assignments

*)
END_FUNCTION_BLOCK

(* @NESTEDCOMMENTS := 'Yes' *)
(* @PATH := '\/Logic\/generators' *)
(* @OBJECTFLAGS := '0, 8' *)
(* @SYMFILEFLAGS := '2048' *)
FUNCTION_BLOCK SCHEDULER_2
VAR_INPUT
	E0 : BOOL;
	E1 : BOOL;
	E2 : BOOL;
	E3 : BOOL;
END_VAR
VAR_INPUT (* CONSTANT *)
	C0, C1, C2, C3 : UINT;
	O0, O1, O2, O3 : UINT;
END_VAR
VAR_OUTPUT
	Q0, Q1, Q2, Q3 : BOOL;
END_VAR
VAR
	sx : UINT;
END_VAR

(*
version 1.0	29. sep 2008
programmer 	hugo
tested by		tobias

SCHEDULER_2 is used to call programs or function blocks at specific cycles.
C0..C3 defines after how many cycles the output becomes active.
O0..O3 defines a cycle offset at startup.

*)

(* @END_DECLARATION := '0' *)
Q0 := E0 AND (sx MOD C0 - O0 = 0);
Q1 := E1 AND (sx MOD C1 - O1 = 0);
Q2 := E2 AND (sx MOD C2 - O2 = 0);
Q3 := E3 AND (sx MOD C3 - O3 = 0);

(* increment cycle counter every cycle *)
sx := sx + 1;

(* revision history
hm 29. sep. 2008		rev 1.0
	original version

*)
END_FUNCTION_BLOCK

(* @NESTEDCOMMENTS := 'Yes' *)
(* @PATH := '\/Logic\/generators' *)
(* @OBJECTFLAGS := '0, 8' *)
(* @SYMFILEFLAGS := '2048' *)
FUNCTION_BLOCK SEQUENCE_4
VAR_INPUT
	in0 : BOOL := TRUE;
	in1 : BOOL := TRUE;
	in2 : BOOL := TRUE;
	in3 : BOOL := TRUE;
	start : BOOL;
	rst : BOOL;
	wait0 : TIME;
	delay0 : TIME;
	wait1 : TIME;
	delay1 : TIME;
	wait2 : TIME;
	delay2 : TIME;
	wait3 : TIME;
	delay3 : TIME;
END_VAR
VAR_INPUT (* CONSTANT *)
	stop_on_error : BOOL;
END_VAR
VAR_OUTPUT
	Q0 : BOOL;
	Q1 : BOOL;
	Q2 : BOOL;
	Q3 : BOOL;
	QX : BOOL;
	run: BOOL;
	step : INT := -1;
	status : BYTE;
END_VAR
VAR
	last : TIME;
	edge : BOOL;
	tx: TIME;
	init: BOOL;
END_VAR

(*
version 1.5	13. mar. 2009
programmer 	oscat
tested by		hans

sequence_4 enables run when a low to high transition is present on start.
a low to high transition on start will restart the sequencer at any time while a rst will hold the sequencer in reset while true.
after run is enabled with a rising edge on start the sequencer waits for wait0 on in0 to enable q0 which stays on for delay0.
the next cycle starts with wait1, continues with delay 1 and so on...
if an edge is not detected during the wait period, the sequencer will then display the error number on the status output.
the status numbers 1..4 are errors in step 0..3.
after the last step that sets q3, the sequencer leaves q3 on for delay3 and then resets to the initial state.
a step output will indicate the current step of the sequencer and will also be present with a fault condition.
after the first output is turened on the sequencer switches from q0 to q1 and so on, at any time there is only one output enabled.
if an input signal is not detected during a wait period, the sequencer will display the error number ( 1 for in0, 2 for in1 .... ).
when an error is present and the config variable stop_on_error is set then the sequencer will stop. otherwise it will continue.
The status output will also display 110 for waiting and 111 for sequence running.
*)
(* @END_DECLARATION := '0' *)
(* read sps timer *)
tx := DWORD_TO_TIME(T_PLC_MS());

(* initialize on startup *)
IF NOT init THEN
	last := tx;
	init := TRUE;
	status := 110;
END_IF;

(* asynchronous reset *)
IF rst THEN
	step := -1;
	Q0 := 0;
	Q1 := 0;
	Q2 := 0;
	Q3 := 0;
	status := 110;
	run := 0;

(* edge on start input restarts the sequencer *)
ELSIF start AND NOT edge THEN
	step := 0;
	last := tx;
	status := 111;
	Q0 := 0;
	Q1 := 0;
	Q2 := 0;
	Q3 := 0;
	run := 1;
END_IF;
edge := start;

(* check if stop on status is necessary *)
IF status > 0 AND status < 100 AND stop_on_error THEN RETURN; END_IF;

(* sequence is running *)
IF run AND step = 0 THEN
	IF NOT q0 AND in0 AND tx - last <= wait0 THEN
		Q0 := TRUE;
		last := tx;
	ELSIF NOT q0 AND tx - last > wait0 THEN
		status := 1;
		run := FALSE;
	ELSIF q0 AND tx - last >= delay0 THEN
		step := 1;
		last := tx;
	END_IF;
END_IF;
IF run AND step = 1 THEN
	IF NOT q1 AND in1 AND tx - last <= wait1 THEN
		Q0 := FALSE;
		Q1 := TRUE;
		last := tx;
	ELSIF NOT q1 AND Tx - last > wait1 THEN
		status := 2;
		q0 := FALSE;
		run := FALSE;
	ELSIF q1 AND tx - last >= delay1 THEN
		step := 2;
		last := tx;
	END_IF;
END_IF;
IF run AND step = 2 THEN
	IF NOT q2 AND in2 AND tx - last <= wait2 THEN
		Q1 := FALSE;
		Q2 := TRUE;
		last := tx;
	ELSIF NOT q2 AND Tx - last > wait2 THEN
		status := 3;
		q1 := FALSE;
		run := FALSE;
	ELSIF q2 AND tx - last >= delay2 THEN
		step := 3;
		last := tx;
	END_IF;
END_IF;
IF run AND step = 3 THEN
	IF NOT q3 AND in3 AND tx - last <= wait3 THEN
		Q2 := FALSE;
		Q3 := TRUE;
		last := tx;
	ELSIF NOT q3 AND Tx - last > wait3 THEN
		status := 4;
		q2 := FALSE;
		run := FALSE;
	ELSIF q3 AND tx - last >= delay3 THEN
		step := -1;
		q3 := FALSE;
		run := FALSE;
		status := 110;
	END_IF;
END_IF;
QX := q0 OR q1 OR q2 OR q3;

(*
hm 1.10.06		rev 1.1
	corrected delay logic to be after event and not before
	added any output

hm 1.12.06		rev 1.2
	corrected failure in sequence logic.
	added init at startup to prevent from initial error after start.

hm 17.1.2007		rev 1.3
	changed output fault to status for better compatibility with other modules (ESR).
	added stop on error functionality and setup variable
	default for inputs in0..3 is true.
	renamed variable state to step

hm	17.sep 2007	rev 1.4
	replaced time() with T_PLC_MS() for compatibility reasons

hm	13. mar. 2009	rev 1.5
	renamed output any to qx for compatibility resons

*)
END_FUNCTION_BLOCK

(* @NESTEDCOMMENTS := 'Yes' *)
(* @PATH := '\/Logic\/generators' *)
(* @OBJECTFLAGS := '0, 8' *)
(* @SYMFILEFLAGS := '2048' *)
FUNCTION_BLOCK SEQUENCE_64
VAR_INPUT
	START : BOOL;
	SMAX : INT;
	PROG : ARRAY[0..63]OF TIME;
	RST : BOOL;
END_VAR
VAR_OUTPUT
	STATE : INT := -1;
	TRIG : BOOL;
END_VAR
VAR
	tx : TIME;
	edge: BOOL;
	last: TIME;
END_VAR

(*
version 1.0	29. jun. 2008
programmer 	hugo
tested by	oscat

sequence generates a sequence of states with a programmable length for each state.

*)

(* @END_DECLARATION := '0' *)
(* read system timer *)
tx := DWORD_TO_TIME(T_PLC_MS());
TRIG := FALSE;

IF RST THEN
	STATE := -1;

(* start sequence *)
ELSIF START AND NOT edge THEN
	STATE := 0;
	last := tx;
	TRIG := TRUE;

(* sequence generator *)
ELSIF (STATE >= 0) THEN
	IF (tx - last) >= PROG[STATE] THEN
		STATE := INC2(STATE, 1, -1, SMAX);
		last := tx;
		TRIG := TRUE;
	END_IF;
END_IF;

edge := START;

(* revision history
hm	29. jun. 2008
	original version

*)
END_FUNCTION_BLOCK

(* @NESTEDCOMMENTS := 'Yes' *)
(* @PATH := '\/Logic\/generators' *)
(* @OBJECTFLAGS := '0, 8' *)
(* @SYMFILEFLAGS := '2048' *)
FUNCTION_BLOCK SEQUENCE_8
VAR_INPUT
	in0 : BOOL := TRUE;
	in1 : BOOL := TRUE;
	in2 : BOOL := TRUE;
	in3 : BOOL := TRUE;
	in4 : BOOL := TRUE;
	in5 : BOOL := TRUE;
	in6 : BOOL := TRUE;
	in7 : BOOL := TRUE;
	start : BOOL;
	rst : BOOL;
	wait0 : TIME;
	delay0 : TIME;
	wait1 : TIME;
	delay1 : TIME;
	wait2 : TIME;
	delay2 : TIME;
	wait3 : TIME;
	delay3 : TIME;
	wait4 : TIME;
	delay4 : TIME;
	wait5 : TIME;
	delay5 : TIME;
	wait6 : TIME;
	delay6 : TIME;
	wait7 : TIME;
	delay7 : TIME;
END_VAR
VAR_INPUT (* CONSTANT *)
	stop_on_error : BOOL;
END_VAR
VAR_OUTPUT
	Q0 : BOOL;
	Q1 : BOOL;
	Q2 : BOOL;
	Q3 : BOOL;
	Q4 : BOOL;
	Q5 : BOOL;
	Q6 : BOOL;
	Q7 : BOOL;
	QX : BOOL;
	run: BOOL;
	step : INT := -1;
	status : BYTE;
END_VAR
VAR
	last : TIME;
	edge : BOOL;
	tx: TIME;
	init: BOOL;
END_VAR

(*
version 1.5	13. mar. 2009
programmer 	oscat
tested by		hans

sequence_8 enables run when a low to high transition is present on start.
a low to high transition on start will restart the sequencer at any time while a rst will hold the sequencer in reset while true.
after run is enabled with a rising edge on start the sequencer waits for wait0 on in0 to enable q0 which stays on for delay0.
the next cycle starts with wait1, continues with delay 1 and so on...
if an edge is not detected during the wait period, the sequencer will then display the error number on the status output.
The status numbers are 1 .. 8 for erros in step 0..7.
after the last step that sets q7, the sequencer leaves q7 on for delay7 and then resets to the initial state.
a step output will indicate the current step of the sequencer and will also be present with a fault condition.
after the first output is turened on the sequencer switches from q0 to q1 and so on, at any time there is only one output enabled.
if an input signal is not detected during a wait period, the sequencer will display the error number ( 1 for in0, 2 for in1 .... ).
when an error is present and the config variable stop_on_error is set then the sequencer will stop. otherwise it will continue.
The status output will also display 110 for waiting and 111 sequece running.

*)
(* @END_DECLARATION := '0' *)
(* read sps timer *)
tx := DWORD_TO_TIME(T_PLC_MS());

(* initialize on startup *)
IF NOT init THEN
	last := tx;
	init := TRUE;
	status := 110;
END_IF;

(* asynchronous reset *)
IF rst THEN
	step := -1;
	Q0 := 0;
	Q1 := 0;
	Q2 := 0;
	Q3 := 0;
	Q4 := 0;
	Q5 := 0;
	Q6 := 0;
	Q7 := 0;
	status := 110;
	run := 0;

(* edge on start input restarts the sequencer *)
ELSIF start AND NOT edge THEN
	step := 0;
	last := tx;
	status := 111;
	Q0 := 0;
	Q1 := 0;
	Q2 := 0;
	Q3 := 0;
	Q4 := 0;
	Q5 := 0;
	Q6 := 0;
	Q7 := 0;
	run := 1;
END_IF;
edge := start;

(* check if stop on error is necessary *)
IF status > 0 AND status < 100 AND stop_on_error THEN RETURN; END_IF;

(* sequence is running *)
IF run AND step = 0 THEN
	IF NOT q0 AND in0 AND tx - last <= wait0 THEN
		Q0 := TRUE;
		last := tx;
	ELSIF NOT q0 AND tx - last > wait0 THEN
		status := 1;
		run := FALSE;
	ELSIF q0 AND tx - last >= delay0 THEN
		step := 1;
		last := tx;
	END_IF;
END_IF;
IF run AND step = 1 THEN
	IF NOT q1 AND in1 AND tx - last <= wait1 THEN
		Q0 := FALSE;
		Q1 := TRUE;
		last := tx;
	ELSIF NOT q1 AND Tx - last > wait1 THEN
		status := 2;
		q0 := FALSE;
		run := FALSE;
	ELSIF q1 AND tx - last >= delay1 THEN
		step := 2;
		last := tx;
	END_IF;
END_IF;
IF run AND step = 2 THEN
	IF NOT q2 AND in2 AND tx - last <= wait2 THEN
		Q1 := FALSE;
		Q2 := TRUE;
		last := tx;
	ELSIF NOT q2 AND Tx - last > wait2 THEN
		status := 3;
		q1 := FALSE;
		run := FALSE;
	ELSIF q2 AND tx - last >= delay2 THEN
		step := 3;
		last := tx;
	END_IF;
END_IF;
IF run AND step = 3 THEN
	IF NOT q3 AND in3 AND tx - last <= wait3 THEN
		Q2 := FALSE;
		Q3 := TRUE;
		last := tx;
	ELSIF NOT q3 AND Tx - last > wait3 THEN
		status := 4;
		q2 := FALSE;
		run := FALSE;
	ELSIF q3 AND tx - last >= delay3 THEN
		step := 4;
		last := tx;
	END_IF;
END_IF;
IF run AND step = 4 THEN
	IF NOT q4 AND in4 AND tx - last <= wait4 THEN
		Q3 := FALSE;
		Q4 := TRUE;
		last := tx;
	ELSIF NOT q4 AND Tx - last > wait4 THEN
		status := 5;
		q3 := FALSE;
		run := FALSE;
	ELSIF q4 AND tx - last >= delay4 THEN
		step := 5;
		last := tx;
	END_IF;
END_IF;
IF run AND step = 5 THEN
	IF NOT q5 AND in5 AND tx - last <= wait5 THEN
		Q4 := FALSE;
		Q5 := TRUE;
		last := tx;
	ELSIF NOT q5 AND Tx - last > wait5 THEN
		status := 6;
		q4 := FALSE;
		run := FALSE;
	ELSIF q5 AND tx - last >= delay5 THEN
		step := 6;
		last := tx;
	END_IF;
END_IF;
IF run AND step = 6 THEN
	IF NOT q6 AND in6 AND tx - last <= wait6 THEN
		Q5 := FALSE;
		Q6 := TRUE;
		last := tx;
	ELSIF NOT q6 AND Tx - last > wait6 THEN
		status := 7;
		q5 := FALSE;
		run := FALSE;
	ELSIF q6 AND tx - last >= delay6 THEN
		step := 7;
		last := tx;
	END_IF;
END_IF;
IF run AND step = 7 THEN
	IF NOT q7 AND in7 AND tx - last <= wait7 THEN
		Q6 := FALSE;
		Q7 := TRUE;
		last := tx;
	ELSIF NOT q7 AND Tx - last > wait7 THEN
		status := 8;
		q6 := FALSE;
		run := FALSE;
	ELSIF q7 AND tx - last >= delay7 THEN
		step := -1;
		Q7 := FALSE;
		Run := FALSE;
		status := 110;
	END_IF;
END_IF;
QX := q0 OR q1 OR q2 OR q3 OR q4 OR q5 OR q6 OR q7;
